Omron Sysmac Studio project delta_paper_0_2 (Sysmac Studio 1.54.0.64019, StandardProject)
(* parameteriaztion the n *)

# Controller new_Controller_0: NX1P2-1140DT version 1.18
Units and slaves: Node47 : MADLN05BE (E002); Node72 : MADLN05BE (E001); Node73 : MADLN05BE (E003)
Axis MC_Axis1, settings changed from default: AxisType=ServoType, UnitsConversion=EnumElement5, UnitsNumerator=8388608, UnitsDenominator=36, MaxVelocity=500, MaxJogVelocity=360, SoftwareLimitMode=ValidForSpecifiedValueImmediateStop, PositiveSoftwareLimit=75, NegativeSoftwareLimit=-29.2, OriginInputMode=EXT, StartDirection=NegativeDirection, OriginInputDetectionDirection=NegativeDirection, HomingVelocity=100, HomingApproachVelocity=10, HomingAcceleration=10, HomingDeceleration=20
Axis MC_Axis2, settings changed from default: AxisNumber=1, AxisType=ServoType, UnitsConversion=EnumElement5, UnitsNumerator=8388608, UnitsDenominator=36, MaxVelocity=500, MaxJogVelocity=360, SoftwareLimitMode=ValidForSpecifiedValueImmediateStop, PositiveSoftwareLimit=75, NegativeSoftwareLimit=-29.2
Axis MC_Axis3, settings changed from default: AxisNumber=2, AxisType=ServoType, UnitsConversion=EnumElement5, UnitsNumerator=8388608, UnitsDenominator=36, MaxVelocity=500, MaxJogVelocity=360, SoftwareLimitMode=ValidForSpecifiedValueDecreaseStop, PositiveSoftwareLimit=29.2, NegativeSoftwareLimit=-75
Task PrimaryTask (priority 4, period or condition 4000): Program0

TYPE InforRobot : STRUCT
    e : LREAL;
    rf : LREAL;
    re : LREAL;
    f : LREAL;
END_STRUCT END_TYPE
TYPE Input_Position : STRUCT
    X : LREAL;
    Y : LREAL;
    Z : LREAL;
END_STRUCT END_TYPE
TYPE Angle_Theta : STRUCT
    Theta1 : LREAL;
    Theta2 : LREAL;
    Theta3 : LREAL;
END_STRUCT END_TYPE
TYPE Bool_Theta : STRUCT
    Motor_Theta1 : REAL;
    Motor_Theta2 : REAL;
    Motor_Theta3 : REAL;
END_STRUCT END_TYPE
TYPE Speed_Theta : STRUCT
    Speed_Theta1 : REAL;
    Speed_Theta2 : REAL;
    Speed_Theta3 : REAL;
END_STRUCT END_TYPE
TYPE Workspace : STRUCT
    X_Min : REAL;
    X_Max : REAL;
    Y_Min : REAL;
    Y_Max : REAL;
    Z_Min : REAL;
    Z_Max : REAL;
END_STRUCT END_TYPE
TYPE From_pc : STRUCT
    n_points : INT;  (* new-> # of points *)
    commandID : INT;
    argument_number : INT;
    argument_x : ARRAY[0..31] OF real;
    argument_y : ARRAY[0..31] OF real;
    argument_z : ARRAY[0..31] OF real;
    argument_e : ARRAY[0..31] OF int;
    bit_doing : INT;
END_STRUCT END_TYPE
TYPE From_plc : STRUCT
    pos_angular : ARRAY[0..2] OF REAL;
    pos_EE : ARRAY[0..6] OF REAL;
    task_doing : INT;
    task_state : INT;
    Total_Time_Estimate : ARRAY[0..30] OF REAL;
    Total_Time_Sum : REAL;
    current_step : INT;
    n_points_ack : INT;
END_STRUCT END_TYPE

VAR_GLOBAL CONSTANT
    MC_Axis1 : _sAXIS_REF;  (* at MC://_MC_AX[0] *)
    MC_Axis2 : _sAXIS_REF;  (* at MC://_MC_AX[1] *)
    MC_Axis3 : _sAXIS_REF;  (* at MC://_MC_AX[2] *)
END_VAR
VAR_GLOBAL
    Out_Test0 : LREAL;
    Out_TestAngle1 : LREAL;
    Out_TestAngle2 : LREAL;
    Out_TestAngle3 : LREAL;
    MyHomingPara : _sHOMING_REF;
    Home_Axis1 : BOOL;  (* at BuiltInIO://cpu/#0/Input_Bit_00 *)
    Home_Axis2 : BOOL;  (* at BuiltInIO://cpu/#0/Input_Bit_01 *)
    Home_Axis3 : BOOL;  (* at BuiltInIO://cpu/#0/Input_Bit_02 *)
    Home_Lamp1 : BOOL;  (* at BuiltInIO://cpu/#0/Output_Bit_00 *)
    Home_Lamp2 : BOOL;  (* at BuiltInIO://cpu/#0/Output_Bit_01 *)
    Home_Lamp3 : BOOL;  (* at BuiltInIO://cpu/#0/Output_Bit_02 *)
    Out_Done_Inter : BOOL;
    pc_package : From_pc;  (* published *)
    plc_package : From_plc;  (* published *)
    Pump_Out : BOOL;  (* at BuiltInIO://cpu/#0/Output_Bit_03 *)
    Mc_On_Btn : BOOL;  (* at BuiltInIO://cpu/#0/Input_Bit_03 *)
    Res_Err_Btn : BOOL;  (* at BuiltInIO://cpu/#0/Input_Bit_04 *)
    Valve_Out : BOOL;  (* at BuiltInIO://cpu/#0/Output_Bit_04 *)
    Start_Home_Flag : BOOL;
    Home_Done_Flag1 : BOOL;
    Home_Done_Flag2 : BOOL;
    Home_Done_Flag3 : BOOL;
    button_teaching_ex : BOOL;  (* at BuiltInIO://cpu/#0/Input_Bit_06 *)
END_VAR
VAR_GLOBAL CONSTANT
    ICV_MAX_PT : UINT := 32;
END_VAR
VAR_GLOBAL
    ICV_n : INT := 4;
    ICV_Abort : BOOL;  (* Huy quy dao giua chung - noi tu Rung 1 E-Stop *)
    ICV_Err_Reset : BOOL;
    ICV_Pos_X : ARRAY[0..31] OF Lreal;
    ICV_Pos_Y : ARRAY[0..31] OF Lreal;
    ICV_Pos_Z : ARRAY[0..31] OF Lreal;
END_VAR

PROGRAM Program0
VAR
    Pw_servo_on : BOOL := False;
    MC_Move_Abs : BOOL;
    Pw_Power_0 : MC_Power;
    Pw_Power_1 : MC_Power;
    Pw_Power_2 : MC_Power;
    MC_Home_Ext : BOOL;  (* toggle 1 *)
    MC_Home_Delta_0 : MC_Home_Delta;
    Calib_Abs1 : MC_MoveAbsolute;
    Calib_Abs2 : MC_MoveAbsolute;
    Calib_Abs3 : MC_MoveAbsolute;
    Home_test_1 : MC_Home;
    Home_test_2 : MC_Home;
    Home_test_3 : MC_Home;
    X_cal : LREAL;
    Y_cal : LREAL;
    Z_cal : LREAL;
    pos_angular : LREAL;
    Goto_Abs : Goto_Absolute;
    when_it_turn2 : BOOL;
    Goto_abs_x : LREAL;
    Goto_abs_y : LREAL;
    Goto_abs_z : LREAL;
    another4 : BOOL;
    MC_Inter_Curve_Vel_0 : MC_Inter_Curve_Vel;
    MC_Inter_Curve_Vel_1 : MC_Inter_Curve_Vel;
    MC_Inter_Curve_Vel_2 : MC_Inter_Curve_Vel;
    MC_Inter_Curve_Vel_3 : MC_Inter_Curve_Vel;
    MC_Inter_Curve_Vel_4 : MC_Inter_Curve_Vel;
    MC_Inter_Curve_Vel_5 : MC_Inter_Curve_Vel;
    ICV_Start_NewTurn : BOOL;  (* Set 1 until ICV_Blend_done_2 *)
    ICV_Vmax : LREAL := 300;  (* 300 *)
    ICV_Amax : LREAL := 1000;  (* 1000 *)
    ICV_Dmax : LREAL := 1000;  (* 1000 *)
    Pump_Ext : BOOL;
    ICV_Pos_E : ARRAY[0..31] OF Int;
    ICV_t : ARRAY[0..30] OF Lreal;
    i1 : INT;
    MC_Goto_Abs : BOOL;  (* Set 1 until it done *)
    Fwk_Calc_OutX : REAL;
    Fwk_Calc_OutY : REAL;
    Fwk_Calc_OutZ : REAL;
    Moveto_Intermediary : MC_MoveAbsolute;
    Moveto_Midpoint : MC_MoveAbsolute;
    Moveto_Midpoint_1 : MC_MoveAbsolute;
    Moveto_Midpoint_2 : MC_MoveAbsolute;
    Moveto_Midpoint_3 : MC_MoveAbsolute;
    Home_Done : BOOL;
    Home_Error : BOOL;
    Goto_Abs_Error : BOOL;
    Pump_Res : BOOL;
    MC_ICV_Err : BOOL;
    MC_Stop1 : MC_Stop;
    MC_Stop2 : MC_Stop;
    MC_Stop3 : MC_Stop;
    MC_RES_DB1 : MC_Reset;
    MC_RES_DB2 : MC_Reset;
    MC_RES_DB3 : MC_Reset;
    Comment : BOOL;
    Mc_On_Btn_Flag : BOOL;
    Check_IK : BOOL;
    Goto_Abs2 : Goto_Absolute;
    Goto_Abs2_Exe : BOOL;
    Goto_Abs2_Done : BOOL;
    Out_TestAngle1_tmp : LREAL;
    Out_TestAngle2_tmp : LREAL;
    Out_TestAngle3_tmp : LREAL;
    Out_TestAngle10 : LREAL;
    Out_TestAngle20 : LREAL;
    Out_TestAngle30 : LREAL;
    Stop1 : MC_Power;
    MC_Stop4 : MC_Stop;
    MC_Stop5 : MC_Stop;
    MC_Stop6 : MC_Stop;
    Comment0 : BOOL;
    MC_Inter_Curve_Vel_6 : MC_Inter_Curve_Vel;
    ICV_Blend_Done_6 : BOOL;
    ICV_Vend_6 : LREAL;
    Current_Step : INT;
    fb_PumpTimer : TP;
    Var_Timer_IN : BOOL;
    Timing_for_EEF : TIME;
    i_t : INT;
    Mem_ICV_t5 : LREAL;
    k_t : LREAL;
    Teach_Index : INT := 0;  (* Chỉ số điểm học hiện tại (0..99) *)
    Teach_Max_Points : INT := 100;
    Teach_Array_X : ARRAY[0..99] OF LREAL := [100(0.0)];
    Teach_Array_Y : ARRAY[0..99] OF LREAL := [100(0.0)];
    Teach_Array_Z : ARRAY[0..99] OF LREAL := [100(0.0)];
    Teach_Array_Th1 : ARRAY[0..99] OF LREAL := [100(0.0)];
    Teach_Array_Th2 : ARRAY[0..99] OF LREAL := [100(0.0)];
    Teach_Array_Th3 : ARRAY[0..99] OF LREAL := [100(0.0)];
    Teach_Array_Full_E : BOOL;
    Teach_FB : FB_TeachingMode;
    button_teaching_active : BOOL;
    Traj : FB_ICV_Sequencer;
    ICV_Abort : BOOL := False;
    ICV_Err_Reset : BOOL := False;
    Mem_T_LastSeg : LREAL := 0.0;  (* Chot thoi gian doan cuoi cho bo dinh thoi bom *)
    Seq_LastSegReady : BOOL := False;  (* Doan cuoi VA da tinh xong thoi gian -> moi cho timer bom chay *)
END_VAR
VAR_EXTERNAL
    Out_Test0 : LREAL;
    Out_TestAngle1 : LREAL;
    Out_TestAngle2 : LREAL;
    Out_TestAngle3 : LREAL;
END_VAR
VAR_EXTERNAL CONSTANT
    MC_Axis1 : _sAXIS_REF;
    MC_Axis2 : _sAXIS_REF;
    MC_Axis3 : _sAXIS_REF;
END_VAR
VAR_EXTERNAL
    Home_Axis2 : BOOL;
    Home_Axis3 : BOOL;
    Out_Done_Inter : BOOL;
    plc_package : From_plc;
    pc_package : From_pc;
    Pump_Out : BOOL;
    Home_Axis1 : BOOL;
    Mc_On_Btn : BOOL;
    Res_Err_Btn : BOOL;
    Valve_Out : BOOL;
    Start_Home_Flag : BOOL;
    Home_Done_Flag1 : BOOL;
    Home_Done_Flag2 : BOOL;
    Home_Done_Flag3 : BOOL;
    button_teaching_ex : BOOL;
    ICV_Pos_X : ARRAY[0..31] OF Lreal;
    ICV_Pos_Y : ARRAY[0..31] OF Lreal;
    ICV_Pos_Z : ARRAY[0..31] OF Lreal;
    ICV_n : INT;
END_VAR
VAR
    _p1 : BOOL;
    _t2 : BOOL;
    _t3 : BOOL;
END_VAR

(* Section Section0: ladder, written here as Structured Text *)

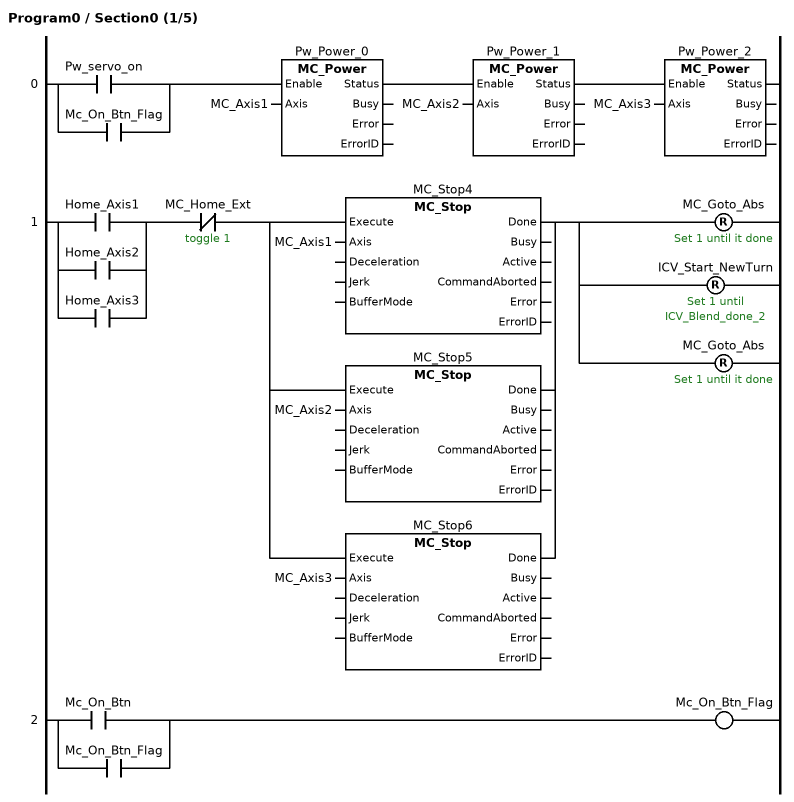
(* Rung 0 *)
Pw_Power_0(Enable := Pw_servo_on OR Mc_On_Btn_Flag, Axis := MC_Axis1);
Pw_Power_1(Enable := Pw_Power_0.Status, Axis := MC_Axis2);
Pw_Power_2(Enable := Pw_Power_1.Status, Axis := MC_Axis3);
(* Rung 1 *)
_p1 := (Home_Axis1 OR Home_Axis2 OR Home_Axis3) AND NOT MC_Home_Ext;
MC_Stop4(Execute := _p1, Axis := MC_Axis1);
MC_Stop5(Execute := _p1, Axis := MC_Axis2);
MC_Stop6(Execute := _p1, Axis := MC_Axis3);
IF MC_Stop4.Done OR MC_Stop5.Done OR MC_Stop6.Done THEN
    MC_Goto_Abs := FALSE;
    ICV_Start_NewTurn := FALSE;
    MC_Goto_Abs := FALSE;
END_IF;
(* Rung 2 *)
Mc_On_Btn_Flag := Mc_On_Btn OR Mc_On_Btn_Flag;

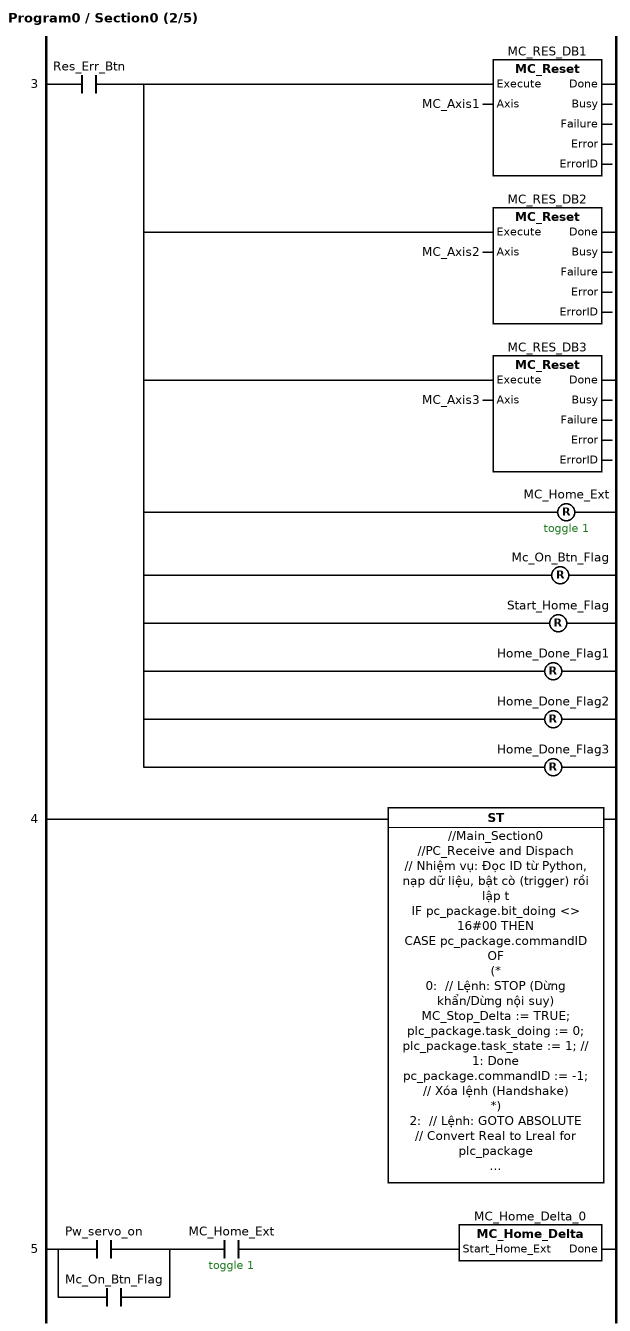
(* Rung 3 *)
MC_RES_DB1(Execute := Res_Err_Btn, Axis := MC_Axis1);
MC_RES_DB2(Execute := Res_Err_Btn, Axis := MC_Axis2);
MC_RES_DB3(Execute := Res_Err_Btn, Axis := MC_Axis3);
IF Res_Err_Btn THEN
    MC_Home_Ext := FALSE;
    Mc_On_Btn_Flag := FALSE;
    Start_Home_Flag := FALSE;
    Home_Done_Flag1 := FALSE;
    Home_Done_Flag2 := FALSE;
    Home_Done_Flag3 := FALSE;
END_IF;
(* Rung 4 *)
//Main_Section0 
//PC_Receive and Dispach
// Nhiệm vụ: Đọc ID từ Python, nạp dữ liệu, bật cò (trigger) rồi lập tức xóa ID

IF pc_package.bit_doing <> 16#00 THEN
CASE pc_package.commandID OF
  (*  
0:  // Lệnh: STOP (Dừng khẩn/Dừng nội suy)
	        MC_Stop_Delta := TRUE;
	        
	        plc_package.task_doing := 0;
	        plc_package.task_state := 1; // 1: Done
	        pc_package.commandID := -1;  // Xóa lệnh (Handshake)
			*)
    2:  // Lệnh: GOTO ABSOLUTE
		// Convert Real to Lreal for plc_package
		Goto_abs_x:= REAL_TO_LREAL(pc_package.argument_x[0]);
		Goto_abs_y := REAL_TO_LREAL(pc_package.argument_y[0]);
		Goto_abs_z:= REAL_TO_LREAL(pc_package.argument_z[0]);
        
        MC_Goto_Abs := TRUE;         // Bật cò chạy
        plc_package.task_doing := 2;
        plc_package.task_state := 2; // 2: Busy
        pc_package.commandID := -1;

    3:  // Lệnh: GO TRAJECTORY (Chạy quỹ đạo theo mảng tọa độ)
        ICV_Start_NewTurn := TRUE; //auto turn off
        FOR i1 := 0 TO 6 DO
			ICV_Pos_X[i1] := REAL_TO_LREAL(pc_package.argument_x[i1]);
			ICV_Pos_Y[i1] := REAL_TO_LREAL(pc_package.argument_y[i1]);
			ICV_Pos_Z[i1] := REAL_TO_LREAL(pc_package.argument_z[i1]);
			ICV_Pos_E[i1] := pc_package.argument_e[i1];
		END_FOR;
        plc_package.task_doing := 3;
        plc_package.task_state := 2; // Busy
        pc_package.commandID := -1;

    4:  // Lệnh: HOME CALIBRATION (Tìm gốc)
        MC_Home_Ext := TRUE;
        
        plc_package.task_doing := 4;
        plc_package.task_state := 2; // Busy
        pc_package.commandID := -1;

    5:  // Lệnh: PICK (Hút vật)
        Pump_Ext := TRUE;
        
        plc_package.task_doing := 5;
        plc_package.task_state := 1; // 1: Done (Do bật bơm là xong ngay)
        pc_package.commandID := -1;

    6:  // Lệnh: RELEASE (Nhả vật)
        Pump_Ext := FALSE;
        
        plc_package.task_doing := 6;
        plc_package.task_state := 1; // Done
        pc_package.commandID := -1;
		END_CASE;
pc_package.bit_doing :=16#00;
END_IF;
(* Rung 5 *)
MC_Home_Delta_0(Start_Home_Ext := (Pw_servo_on OR Mc_On_Btn_Flag) AND MC_Home_Ext);

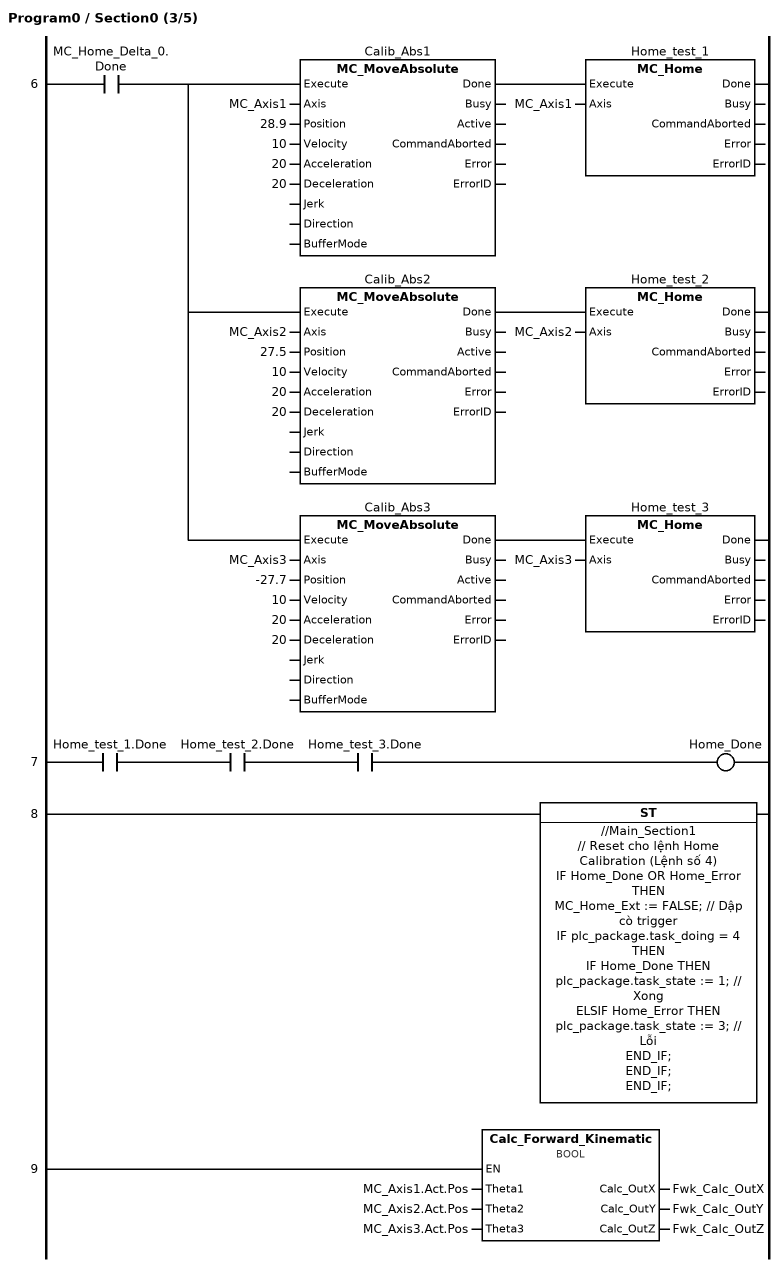
(* Rung 6 *)
Calib_Abs1(Execute := MC_Home_Delta_0.Done, Axis := MC_Axis1, Position := 28.9, Velocity := 10, Acceleration := 20, Deceleration := 20);
Home_test_1(Execute := Calib_Abs1.Done, Axis := MC_Axis1);
Calib_Abs2(Execute := MC_Home_Delta_0.Done, Axis := MC_Axis2, Position := 27.5, Velocity := 10, Acceleration := 20, Deceleration := 20);
Home_test_2(Execute := Calib_Abs2.Done, Axis := MC_Axis2);
Calib_Abs3(Execute := MC_Home_Delta_0.Done, Axis := MC_Axis3, Position := -27.7, Velocity := 10, Acceleration := 20, Deceleration := 20);
Home_test_3(Execute := Calib_Abs3.Done, Axis := MC_Axis3);
(* Rung 7 *)
Home_Done := Home_test_1.Done AND Home_test_2.Done AND Home_test_3.Done;
(* Rung 8 *)
//Main_Section1 
// Reset cho lệnh Home Calibration (Lệnh số 4)
IF Home_Done OR Home_Error THEN
 
    MC_Home_Ext := FALSE; // Dập cò trigger
	
    IF plc_package.task_doing = 4 THEN
        IF Home_Done THEN
            plc_package.task_state := 1; // Xong
        ELSIF Home_Error THEN
            plc_package.task_state := 3; // Lỗi
        END_IF;
    END_IF;
    
END_IF;
(* Rung 9 *)
_t2 := Calc_Forward_Kinematic(Theta1 := MC_Axis1.Act.Pos, Theta2 := MC_Axis2.Act.Pos, Theta3 := MC_Axis3.Act.Pos, Calc_OutX => Fwk_Calc_OutX, Calc_OutY => Fwk_Calc_OutY, Calc_OutZ => Fwk_Calc_OutZ);

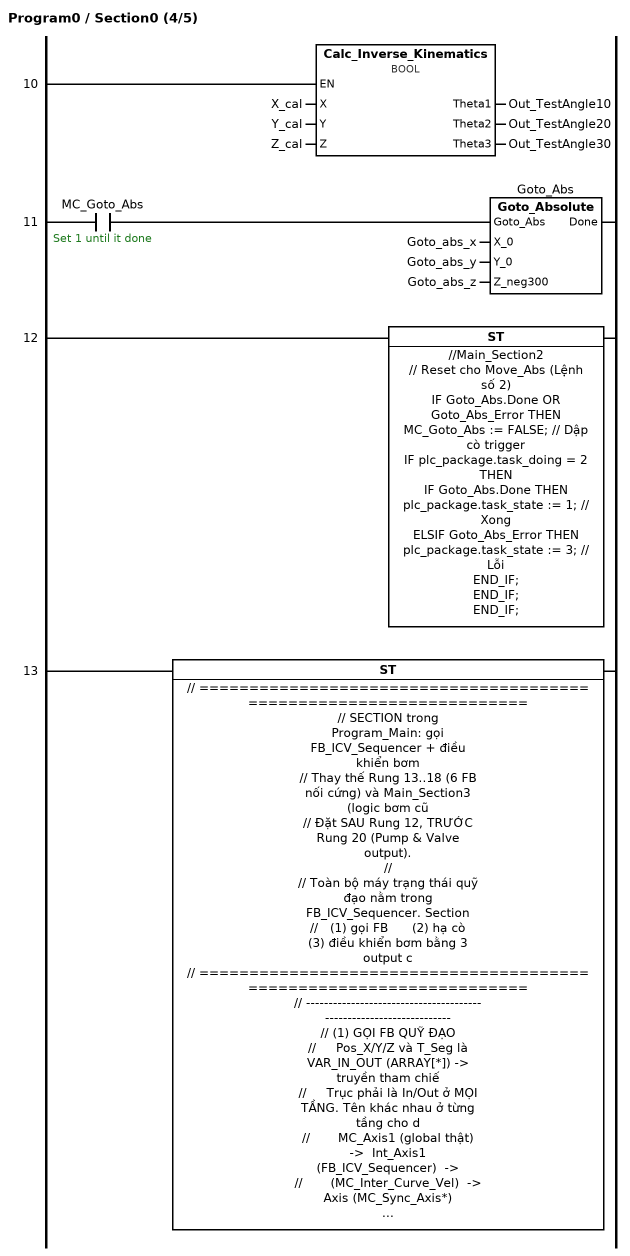
(* Rung 10 *)
_t3 := Calc_Inverse_Kinematics(X := X_cal, Y := Y_cal, Z := Z_cal, Theta1 => Out_TestAngle10, Theta2 => Out_TestAngle20, Theta3 => Out_TestAngle30);
(* Rung 11 *)
Goto_Abs(Goto_Abs := MC_Goto_Abs, X_0 := Goto_abs_x, Y_0 := Goto_abs_y, Z_neg300 := Goto_abs_z);
(* Rung 12 *)
//Main_Section2
// Reset cho Move_Abs (Lệnh số 2)
IF Goto_Abs.Done OR Goto_Abs_Error THEN
 
    MC_Goto_Abs := FALSE; // Dập cò trigger
	
    IF plc_package.task_doing = 2 THEN
        IF Goto_Abs.Done THEN
            plc_package.task_state := 1; // Xong
        ELSIF Goto_Abs_Error THEN
            plc_package.task_state := 3; // Lỗi
        END_IF;
    END_IF;
    
END_IF;
(* Rung 13 *)
// =====================================================================================
// SECTION trong Program_Main: gọi FB_ICV_Sequencer + điều khiển bơm
// Thay thế Rung 13..18 (6 FB nối cứng) và Main_Section3 (logic bơm cũ).
// Đặt SAU Rung 12, TRƯỚC Rung 20 (Pump & Valve output).
//
// Toàn bộ máy trạng thái quỹ đạo nằm trong FB_ICV_Sequencer. Section này chỉ:
//   (1) gọi FB      (2) hạ cò      (3) điều khiển bơm bằng 3 output của FB
// =====================================================================================


// -------------------------------------------------------------------------------------
// (1) GỌI FB QUỸ ĐẠO
//     Pos_X/Y/Z và T_Seg là VAR_IN_OUT (ARRAY[*]) -> truyền tham chiếu, KHÔNG copy mảng.
//     Trục phải là In/Out ở MỌI TẦNG. Tên khác nhau ở từng tầng cho dễ phân biệt:
//       MC_Axis1 (global thật)  ->  Int_Axis1 (FB_ICV_Sequencer)  ->  MC_Axis1
//       (MC_Inter_Curve_Vel)  ->  Axis (MC_Sync_Axis*)
// -------------------------------------------------------------------------------------
Traj(
    Execute  := ICV_Start_NewTurn,
    Abort    := ICV_Abort,
    ErrReset := ICV_Err_Reset,
    N_Points := ICV_n,
    Max_Index:= 31,                 // chỉ số lớn nhất của ICV_Pos_X (ARRAY[0..31])
    V_max    := ICV_Vmax,
    A_max    := ICV_Amax,
    D_max    := ICV_Dmax,
    Pos_X    := ICV_Pos_X,
    Pos_Y    := ICV_Pos_Y,
    Pos_Z    := ICV_Pos_Z,
    T_Seg    := ICV_t,
    // TRÁI = tên tham số của FB_ICV_Sequencer ; PHẢI = biến global của trục thật
    Int_Axis1:= MC_Axis1,
    Int_Axis2:= MC_Axis2,
    Int_Axis3:= MC_Axis3
);


// -------------------------------------------------------------------------------------
// (2) HẠ CÒ NGAY SAU LỜI GỌI
//     FB đã bắt SƯỜN LÊN của Execute ở khối (1) rồi, nên hạ ngay là an toàn.
//
//     KHÔNG dùng "IF Traj.Busy THEN": khi FB TỪ CHỐI lệnh (N_Points sai -> ErrorID = 1)
//     thì Busy KHÔNG BAO GIỜ lên TRUE -> cò kẹt TRUE vĩnh viễn -> mọi lệnh sau đó không
//     tạo được sườn lên nữa -> quỹ đạo chết hẳn, phải khởi động lại PLC.
// -------------------------------------------------------------------------------------
IF ICV_Start_NewTurn THEN
    ICV_Start_NewTurn := FALSE;
END_IF;

// Xoá cờ ErrReset sau 1 chu kỳ (nút Res_Err_Btn có thể bị giữ lâu)
IF ICV_Err_Reset AND NOT Traj.Error THEN
    ICV_Err_Reset := FALSE;
END_IF;


// -------------------------------------------------------------------------------------
// (3) ĐIỀU KHIỂN BƠM / END-EFFECTOR
//     Đoạn 0 .. n-3 : bơm bám theo ICV_Pos_E[SegIdx]
//     Đoạn cuối     : bơm nhả sớm ở 50% thời gian đoạn, cho vật kịp rơi trước khi tay đi
// -------------------------------------------------------------------------------------

// "Đoạn cuối SẴN SÀNG" = đang ở đoạn cuối VÀ FB đã tính xong thời gian của đoạn đó.
//
// PHẢI chờ T_SegNow > 0. Ngay chu kỳ vừa chuyển sang đoạn cuối, Out_T_Segment của
// MC_Inter_Curve_Vel VẪN ĐANG GIỮ thời gian của đoạn TRƯỚC (nó chỉ bị xoá ở State 0
// của đoạn mới, tức chu kỳ sau). Chốt vội sẽ lấy nhầm số của đoạn trước.
Seq_LastSegReady := Traj.IsLastSeg AND (Traj.T_SegNow > 0.0);

IF Seq_LastSegReady THEN
    Mem_T_LastSeg := Traj.T_SegNow;
END_IF;

Timing_for_EEF := NanoSecToTime(LREAL_TO_LINT(0.5 * Mem_T_LastSeg * 1000000000.0));

// IN dùng Seq_LastSegReady, KHÔNG dùng Traj.IsLastSeg.
// TP chốt PT tại SƯỜN LÊN của IN -> phải đợi PT đúng rồi mới cho timer chạy.
// Trễ 2 chu kỳ (8 ms) so với đầu đoạn cuối, không đáng kể.
fb_PumpTimer(IN := Seq_LastSegReady, PT := Timing_for_EEF);

IF NOT Traj.Busy THEN
    Pump_Ext := FALSE;

ELSIF Traj.IsLastSeg THEN
    // GIỮ NGUYÊN biểu thức của code cũ: đúng khi fb_PumpTimer khai báo là TP (Pulse).
    //   TP  -> .Q = TRUE trong 50% đầu, tự hạ sau đó -> bơm nhả ở giữa đoạn.  ĐÚNG
    //   TON -> .Q = FALSE trong 50% đầu -> bơm chỉ bật ở nửa SAU. NGƯỢC Ý ĐỒ.
    // Nếu instance đang là TON, đổi thành:  AND NOT fb_PumpTimer.Q
    //
    // "OR NOT Seq_LastSegReady" giữ bơm ON trong 2 chu kỳ chờ timer khởi động,
    // tránh hụt chân không 8 ms ngay đầu đoạn cuối.
    Pump_Ext := (ICV_Pos_E[Traj.SegIdx] = 1)
                AND (fb_PumpTimer.Q OR NOT Seq_LastSegReady);

ELSE
    Pump_Ext := (ICV_Pos_E[Traj.SegIdx] = 1);
END_IF;

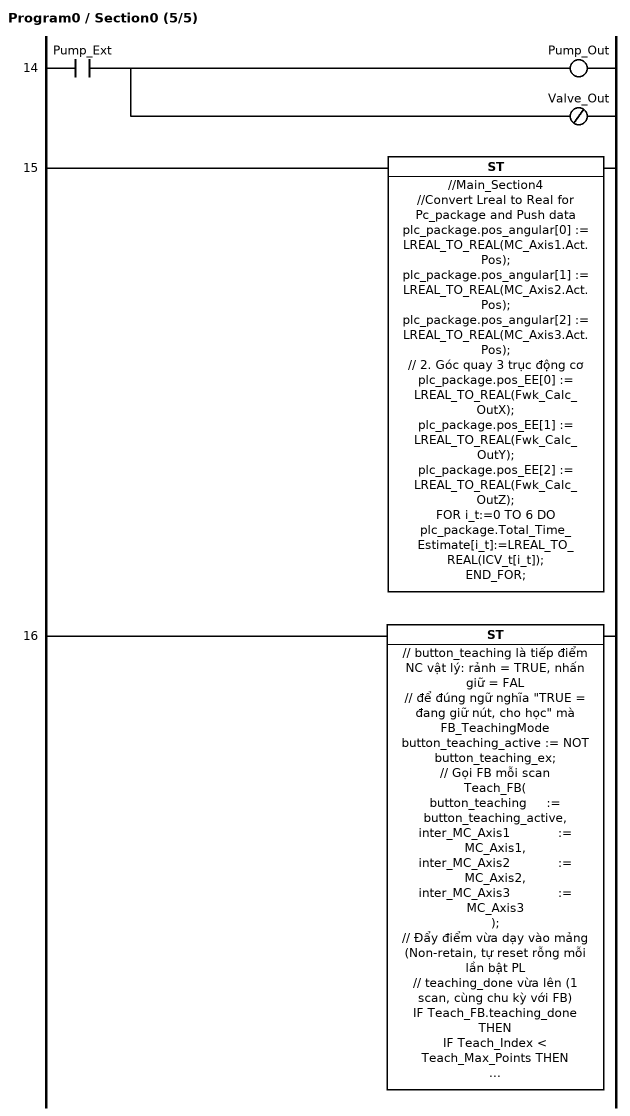
(* Rung 14 *)
Pump_Out := Pump_Ext;
Valve_Out := NOT Pump_Ext;
(* Rung 15 *)
//Main_Section4
//Convert Lreal to Real for Pc_package and Push data
plc_package.pos_angular[0] := LREAL_TO_REAL(MC_Axis1.Act.Pos);
plc_package.pos_angular[1] := LREAL_TO_REAL(MC_Axis2.Act.Pos);
plc_package.pos_angular[2] := LREAL_TO_REAL(MC_Axis3.Act.Pos);

// 2. Góc quay 3 trục động cơ
plc_package.pos_EE[0] := LREAL_TO_REAL(Fwk_Calc_OutX); 
plc_package.pos_EE[1] := LREAL_TO_REAL(Fwk_Calc_OutY); 
plc_package.pos_EE[2] := LREAL_TO_REAL(Fwk_Calc_OutZ);

FOR i_t:=0 TO 6 DO
	plc_package.Total_Time_Estimate[i_t]:=LREAL_TO_REAL(ICV_t[i_t]);
END_FOR;
(* Rung 16 *)
// button_teaching là tiếp điểm NC vật lý: rảnh = TRUE, nhấn giữ = FALSE -> đảo lại
// để đúng ngữ nghĩa "TRUE = đang giữ nút, cho học" mà FB_TeachingMode yêu cầu.
button_teaching_active := NOT button_teaching_ex;

// Gọi FB mỗi scan
Teach_FB(
    button_teaching     := button_teaching_active,
    inter_MC_Axis1            := MC_Axis1,
    inter_MC_Axis2            := MC_Axis2,
    inter_MC_Axis3            := MC_Axis3	
);

// Đẩy điểm vừa dạy vào mảng (Non-retain, tự reset rỗng mỗi lần bật PLC) — chỉ khi
// teaching_done vừa lên (1 scan, cùng chu kỳ với FB)
IF Teach_FB.teaching_done THEN
    IF Teach_Index < Teach_Max_Points THEN
        Teach_Array_X[Teach_Index]   := Teach_FB.pos_teaching1;
        Teach_Array_Y[Teach_Index]   := Teach_FB.pos_teaching2;
        Teach_Array_Z[Teach_Index]   := Teach_FB.pos_teaching3;
        Teach_Array_Th1[Teach_Index] := LREAL_TO_REAL(Teach_FB.theta_teaching1);
        Teach_Array_Th2[Teach_Index] := LREAL_TO_REAL(Teach_FB.theta_teaching2);
        Teach_Array_Th3[Teach_Index] := LREAL_TO_REAL(Teach_FB.theta_teaching3);
        Teach_Index := Teach_Index + 1;
        Teach_Array_Full_E := FALSE;
    ELSE
        // Mảng đã đầy: không có chỗ lưu, báo lỗi rõ ràng thay vì âm thầm bỏ qua
        Teach_Array_Full_E := TRUE;
    END_IF;
END_IF;

// HMI / Python PC (poll chậm qua TCP/IP) nên theo dõi Teach_Index tăng dần
// thay vì bắt xung teaching_done — tránh miss tín hiệu do chu kỳ poll không đồng bộ scan PLC.
END_PROGRAM

FUNCTION Calc_Inverse_Kinematics : BOOL
VAR CONSTANT
    Cos120 : LREAL := -0.5;
    Sin120 : LREAL := 0.8660254037844386;
END_VAR
VAR
    tmp_Theta1 : LREAL;
    tmp_Theta2 : LREAL;
    tmp_Theta3 : LREAL;
    rotate_X2 : LREAL;
    rotate_Y2 : LREAL;
    rotate_X3 : LREAL;
    rotate_Y3 : LREAL;
END_VAR
VAR CONSTANT
    rf : LREAL := 346.4;
    re : LREAL := 86.6;
    f : LREAL := 140;
    e : LREAL := 315;
END_VAR
VAR
    Out_Error_IK : BOOL;
END_VAR
VAR_INPUT
    X : LREAL;
    Y : LREAL;
    Z : LREAL;
END_VAR
VAR_OUTPUT
    Theta1 : LREAL;
    Theta2 : LREAL;
    Theta3 : LREAL;
END_VAR
// Khởi tạo lại cờ báo lỗi ở mỗi đầu chu kỳ quét (Primary Task)
Out_Error_IK := FALSE;

// -----------------------------------------------------------------------
// TÍNH TOÁN THETA 1 (Cánh tay 1 - Không xoay trục)
// -----------------------------------------------------------------------
Calc_Inverse_Kinematics := Calc_Angles_YZ(
    X0 := X, 
    Y0 := Y, 
    Z0 := Z,
    OutTheta => tmp_Theta1
);

	
// [TỐI ƯU B] Xử lý lỗi an toàn: Nếu tính toán IK thất bại (Tọa độ ngoài tầm với)
IF Calc_Inverse_Kinematics = TRUE  OR tmp_Theta1 <-20 THEN
    Out_Error_IK := TRUE; // Bật cờ báo lỗi ra hệ thống
    RETURN;               // Ngắt tính toán ngay lập tức
END_IF;

// [TỐI ƯU A] Truyền thẳng giá trị LREAL nguyên bản xuống Servo, BỎ HÀM ROUND
Theta1 := tmp_Theta1;


// -----------------------------------------------------------------------
// TÍNH TOÁN THETA 2 (Cánh tay 2 - Xoay hệ tọa độ đi -120 độ)
// -----------------------------------------------------------------------
rotate_X2 := X * Cos120 + Y * Sin120;
rotate_Y2 := Y * Cos120 - X * Sin120;

Calc_Inverse_Kinematics := Calc_Angles_YZ(
    X0 := rotate_X2, 
    Y0 := rotate_Y2, 
    Z0 := Z,
    OutTheta => tmp_Theta2
);

IF Calc_Inverse_Kinematics = TRUE OR tmp_Theta2 <-20 THEN
    Out_Error_IK := TRUE;
    RETURN;
END_IF;

Theta2 := tmp_Theta2;


// -----------------------------------------------------------------------
// TÍNH TOÁN THETA 3 (Cánh tay 3 - Xoay hệ tọa độ đi +120 độ)
// -----------------------------------------------------------------------
rotate_X3 := X * Cos120 - Y * Sin120;
rotate_Y3 := Y * Cos120 + X * Sin120;

Calc_Inverse_Kinematics := Calc_Angles_YZ(
    X0 := rotate_X3, 
    Y0 := rotate_Y3, 
    Z0 := Z,
    OutTheta => tmp_Theta3
);

IF Calc_Inverse_Kinematics = TRUE OR tmp_Theta3*-1 >20 THEN
    Out_Error_IK := TRUE;
    RETURN;
END_IF;

Theta3 := tmp_Theta3*-1;
END_FUNCTION

FUNCTION Calc_Angles_YZ : BOOL  (* return true -> False in inverse calc *)
VAR
    tmp_y0 : LREAL;
    a : LREAL;
    b : LREAL;
    d : LREAL;
    yj : LREAL;
    zj : LREAL;
    y1 : LREAL;
    tmp_AnglePi : LREAL;
END_VAR
VAR CONSTANT
    Pi : LREAL := 3.141592653589793;
    Tan30 : LREAL := 0.5773502691896257;
    Base : LREAL := 346.4;
    EndEffector : LREAL := 86.6;
    Bicep : LREAL := 140;
    Forearm : LREAL := 315;
END_VAR
VAR_INPUT
    X0 : LREAL;
    Y0 : LREAL;
    Z0 : LREAL;
END_VAR
VAR_OUTPUT
    OutTheta : LREAL;
END_VAR
(*
// FUNCTION: Calc_Angles_YZ (Cal the inverse in 2D-space)
//All variants use Lreal to uttilize the precision of servo and syns all data

// [] Bẫy lỗi chia cho 0: Nếu tọa độ Z0 = 0 (End-effector nằm ngang với Base)
// Phép tính 'a' và 'b' bên dưới sẽ bị lỗi chia cho 0 làm CPU PLC báo lỗi (Major Fault)
*)
IF Z0 = 0.0 THEN
    Calc_Angles_YZ := TRUE; // turn Error true
    RETURN;
END_IF;

// Calc the Y1 and have temp_y0 (the prosition of the Y0 with Y1)
y1 := -0.5 * Tan30* Base;   // the point of edge of fix-triangle
tmp_y0 := Y0 - (0.5 *Tan30* EndEffector);  // the point of the edge of active-triagle

// we have ellbow (0,yj,zj) is contraint with:
//1. on a circle (0,y1,0) with R = bicep so (yj-y1)^2 + z_j^2 = bicep^2
//2. distance from End-effector (X0, tmp_y0,z0) equal the Forearm so
// X0^2 + (tmp_y0 - yj)^2 + (z-zj)^2 = forearm^2
// mathemitical tranformation we have linear function z with a and b bellow
// zj = a + b*yj => we have zj and we tranfer it to equation 1 and solve the two level function with yj
a := (X0*X0 + tmp_y0 * tmp_y0 + Z0 * Z0 + Bicep * Bicep - Forearm * Forearm - y1 * y1) / (2.0 * Z0);
b := (y1 - tmp_y0) / Z0;

// the delta of two level function with yj
d := - (a + b * y1) * (a + b * y1) + Bicep * (b * b * Bicep + Bicep);

// Kiểm tra xem điểm có tồn tại trong vùng không gian (Workspace) không
IF d < 0.0 THEN
    Calc_Angles_YZ := TRUE; // Trả về lỗi (Điểm không với tới được)
    RETURN;
END_IF;

yj := (y1 - a * b - SQRT(d)) / (b * b + 1.0);
zj := a + b * yj;

tmp_AnglePi := 0.0;
IF yj > y1 THEN
    tmp_AnglePi := 180.0;
END_IF;

// [TỐI ƯU 3] Bẫy lỗi chia cho 0 trong hàm tính góc ATAN
// Khi y1 = yj, phép chia (-zj / (y1 - yj)) sẽ gây lỗi PLC
IF (y1 - yj) = 0.0 THEN
    IF -zj >= 0.0 THEN
        OutTheta := 90.0 + tmp_AnglePi;
    ELSE
        OutTheta := -90.0 + tmp_AnglePi;
    END_IF;
ELSE
    // Tính góc Theta. Sử dụng hằng số '_pi' có sẵn của Sysmac Studio
    OutTheta := 180.0 * ATAN(-zj / (y1 - yj)) / Pi + tmp_AnglePi;
END_IF;

// Trả về FALSE khi tính toán thành công
Calc_Angles_YZ := FALSE;
RETURN;
END_FUNCTION

FUNCTION Calc_Forward_Kinematic : BOOL
VAR
    w : LREAL;
    Cos30 : LREAL := 0.8660254037844386;
    Pi : LREAL := 3.141592653589793;
    Tan30 : LREAL := 0.5773502691896257;
    Sin30 : LREAL := 0.5;
END_VAR
VAR CONSTANT
    Base : LREAL := 346.4;
    EndEffector : LREAL := 86.6;
    Bicep : LREAL := 140;
    Forearm : LREAL := 315;
END_VAR
VAR
    x_j1 : LREAL;
    y_j1 : LREAL;
    z_j1 : LREAL;
    x_j2 : LREAL;
    y_j2 : LREAL;
    z_j2 : LREAL;
    x_j3 : LREAL;
    y_j3 : LREAL;
    z_j3 : LREAL;
    r1 : LREAL;
    r2 : LREAL;
    r3 : LREAL;
    a1 : LREAL;
    a2 : LREAL;
    b1 : LREAL;
    b2 : LREAL;
    demon : LREAL;
    A_quad : LREAL;
    B_quad : LREAL;
    C_quad : LREAL;
    d : LREAL;
    t3 : LREAL;
    t2 : LREAL;
    t1 : LREAL;
    Calc_Forward_Kinematics : BOOL;
    OutX : LREAL;
    OutZ : LREAL;
    OutY : LREAL;
    D1_coeff : LREAL;
    A1_coeff : LREAL;
    B1_coeff : LREAL;
    C1_coeff : LREAL;
    A2_coeff : LREAL;
    B2_coeff : LREAL;
    C2_coeff : LREAL;
    D2_coeff : LREAL;
    det : LREAL;
END_VAR
VAR_INPUT
    Theta1 : LREAL;
    Theta2 : LREAL;
    Theta3 : LREAL;
END_VAR
VAR_OUTPUT
    Calc_OutX : REAL;
    Calc_OutY : REAL;
    Calc_OutZ : REAL;
END_VAR
VAR_EXTERNAL CONSTANT
    MC_Axis1 : _sAXIS_REF;
    MC_Axis2 : _sAXIS_REF;
    MC_Axis3 : _sAXIS_REF;
END_VAR
// =======================================================================
// FUNCTION: Calc_Forward_Kinematics (Tính toán động học thuận Robot Delta 3D)
// Trả về FALSE nếu tính toán thành công, TRUE nếu điểm nằm ngoài vùng làm việc
// =======================================================================
// LẤY GIÁ TRỊ GÓC THỰC TẾ (ACTUAL POSITION) TỪ ENCODER CỦA TRỤC
// =======================================================================
// Chuyển đổi các góc hiện tại từ Độ sang Radian
t1 := Theta1 * Pi / 180.0;
t2 := Theta2 * Pi / 180.0;
t3 := Theta3 * Pi / -180.0;

// Tính toán độ lệch tâm tương đối giữa Base và EndEffector
// (w chính là dịch tâm ngang từ gốc tọa độ đến khớp khuỷu tay nếu chiếu lên mặt phẳng XY)
w := 0.5 * Tan30 * (Base - EndEffector);

// =======================================================================
// BƯỚC 1: Tìm tọa độ không gian (x, y, z) của 3 khớp khuỷu tay (Elbow Joints)
// Hệ tọa độ tiêu chuẩn: Trục 1 nằm dọc theo phần âm của trục Y
// =======================================================================

// Trục 1 (Góc lệch 0 độ so với trục tính toán, xoay về -Y)
x_j1 := 0.0;
y_j1 := -(w + Bicep * COS(t1));
z_j1 := -Bicep * SIN(t1);

// Trục 2 (Xoay +120 độ)
x_j2 := (w + Bicep * COS(t2)) * Cos30;
y_j2 := (w + Bicep * COS(t2)) * Sin30;
z_j2 := -Bicep * SIN(t2);

// Trục 3 (Xoay -120 độ hoặc 240 độ)
x_j3 := -(w + Bicep * COS(t3)) * Cos30;
y_j3 := (w + Bicep * COS(t3)) * Sin30;
z_j3 := -Bicep * SIN(t3);

// =======================================================================
// BƯỚC 2: Giải hệ 3 phương trình mặt cầu có tâm tại các Elbow, bán kính Forearm
// =======================================================================

// =======================================================================
// BƯỚC 2: Giải hệ 3 phương trình mặt cầu (Dạng tổng quát, KHÔNG RÚT GỌN SAI)
// =======================================================================
// BƯỚC 2: Giải hệ 3 phương trình mặt cầu có tâm tại các Elbow (Phiên bản Tổng quát)
// =======================================================================

// Tính tổng bình phương tọa độ của các Elbow
r1 := y_j1 * y_j1 + z_j1 * z_j1;  // x_j1 = 0
r2 := x_j2 * x_j2 + y_j2 * y_j2 + z_j2 * z_j2;
r3 := x_j3 * x_j3 + y_j3 * y_j3 + z_j3 * z_j3;

// Thiết lập các hệ số cho hệ phương trình tuyến tính 2 ẩn (X, Y) theo tham số Z
// Dạng: 
// A1*X + B1*Y = D1 - C1*Z
// A2*X + B2*Y = D2 - C2*Z

A1_coeff := x_j2;                   // Thực chất là (x_j2 - x_j1) nhưng x_j1 = 0
B1_coeff := y_j2 - y_j1;
C1_coeff := z_j2 - z_j1;
D1_coeff := 0.5 * (r2 - r1);

A2_coeff := x_j3;                   // Thực chất là (x_j3 - x_j1) nhưng x_j1 = 0
B2_coeff := y_j3 - y_j1;
C2_coeff := z_j3 - z_j1;
D2_coeff := 0.5 * (r3 - r1);

// Tính định thức (Determinant) của hệ phương trình
det := (A1_coeff * B2_coeff) - (A2_coeff * B1_coeff);

// Bẫy lỗi: Hệ vô nghiệm (Chỉ xảy ra khi 3 khuỷu tay cùng nằm trên 1 đường thẳng)
IF det = 0.0 THEN
    Calc_Forward_Kinematics := TRUE; 
    RETURN;
END_IF;

// Sử dụng quy tắc Cramer để tìm a1, b1 (Cho X) và a2, b2 (Cho Y)
// Để biểu diễn: X0 = a1 + b1*Z0
a1 := (D1_coeff * B2_coeff - D2_coeff * B1_coeff) / det;
b1 := -(C1_coeff * B2_coeff - C2_coeff * B1_coeff) / det;

// Để biểu diễn: Y0 = a2 + b2*Z0
a2 := (A1_coeff * D2_coeff - A2_coeff * D1_coeff) / det;
b2 := -(A1_coeff * C2_coeff - A2_coeff * C1_coeff) / det;

// =======================================================================
// BƯỚC 3: Thay X0, Y0 vào phương trình mặt cầu 1 để tìm Z0
// Tạo thành phương trình bậc 2: A_quad * Z0^2 + B_quad * Z0 + C_quad = 0
// =======================================================================

A_quad := b1 * b1 + b2 * b2 + 1.0;
B_quad := 2.0 * (a1 * b1 + a2 * b2 - b2 * y_j1 - z_j1);
C_quad := a1 * a1 + a2 * a2 - 2.0 * a2 * y_j1 + r1 - (Forearm * Forearm);

// Tính Delta (Discriminant)
d := (B_quad * B_quad) - (4.0 * A_quad * C_quad);

// Kiểm tra xem vị trí các góc hiện tại có tạo ra tọa độ hợp lệ không
IF d < 0.0 THEN
    Calc_Forward_Kinematics := TRUE; // Trả về lỗi: Các khớp không thể kết nối
    RETURN;
END_IF;

// Tính tọa độ trung tâm End-Effector (Z lấy nghiệm có dấu trừ phía trước SQRT 
// vì đặc thù cơ cấu Delta robot làm việc ở nửa dưới trục Z)
OutZ := (-B_quad - SQRT(d)) / (2.0 * A_quad);

// Đẩy ngược Z0 vào hệ số tuyến tính để tìm X0 và Y0
OutX := a1 + b1 * OutZ;
OutY := a2 + b2 * OutZ;

Calc_OutZ := LREAL_TO_REAL(OutZ);
Calc_OutX := LREAL_TO_REAL(a1 + b1 * OutZ);
Calc_OutY := LREAL_TO_REAL(a2 + b2 * OutZ);

// Tính toán thành công
Calc_Forward_Kinematics := FALSE;
RETURN;
END_FUNCTION

FUNCTION_BLOCK MC_Home_Delta
VAR
    Move_Vel_Axis1 : MC_MoveVelocity;
    Start_Home : BOOL;
    MC_Stop_Axis1 : MC_Stop;
    Move_Vel_Axis2 : MC_MoveVelocity;
    Move_Vel_Axis3 : MC_MoveVelocity;
    MC_Stop_Axis2 : MC_Stop;
    MC_Stop_Axis3 : MC_Stop;
    MC_Home_Axis1 : MC_Home;
    MC_Home_Axis2 : MC_Home;
    MC_Home_Axis3 : MC_Home;
    t_home : TON;
    t2 : TON;
    t1 : TON;
    t3 : TON;
    TP1 : TP;
    TP2 : TP;
    TP4 : TP;
END_VAR
VAR_INPUT
    Start_Home_Ext : BOOL;
END_VAR
VAR_OUTPUT
    Done : BOOL;
END_VAR
VAR_EXTERNAL
    Home_Axis1 : BOOL;
    Home_Axis2 : BOOL;
    Home_Axis3 : BOOL;
END_VAR
VAR_EXTERNAL CONSTANT
    MC_Axis3 : _sAXIS_REF;
    MC_Axis2 : _sAXIS_REF;
    MC_Axis1 : _sAXIS_REF;
END_VAR
VAR_EXTERNAL
    Home_Lamp3 : BOOL;
    Home_Lamp1 : BOOL;
    Home_Lamp2 : BOOL;
    Start_Home_Flag : BOOL;
    Home_Done_Flag1 : BOOL;
    Home_Done_Flag2 : BOOL;
    Home_Done_Flag3 : BOOL;
END_VAR
VAR
    _e1 : R_TRIG;
    _e2 : R_TRIG;
    _e3 : R_TRIG;
    _e4 : R_TRIG;
END_VAR
(* ladder, written here as Structured Text *)

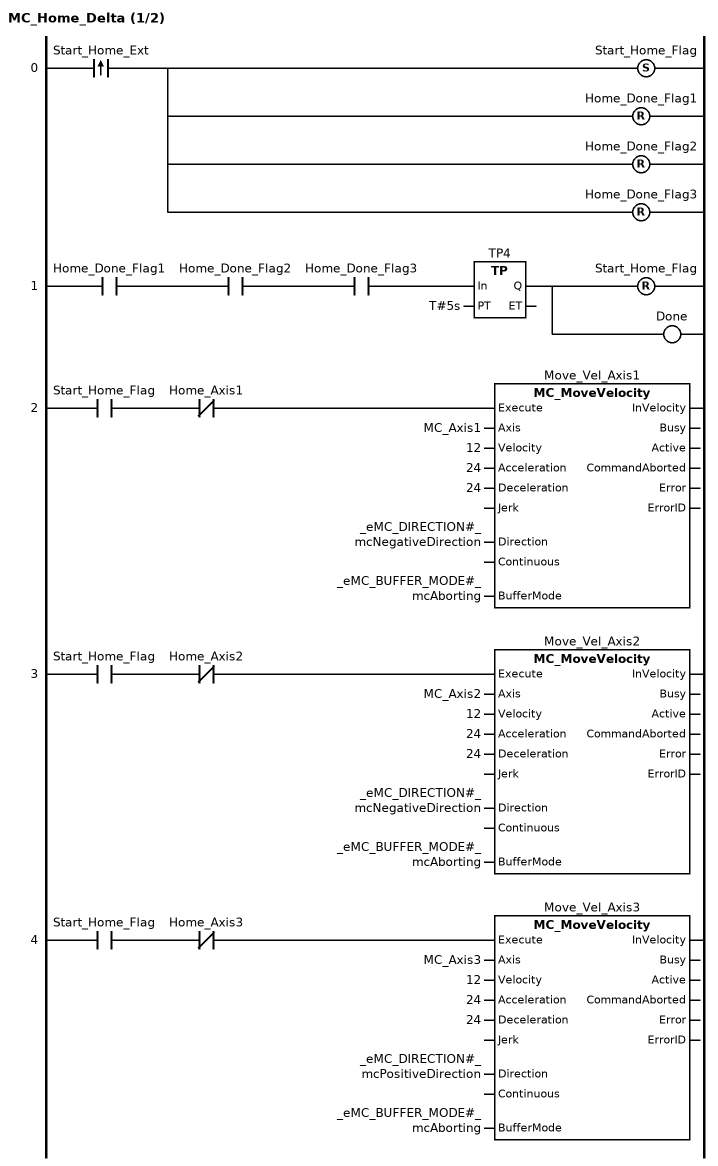
(* Rung 0 *)
_e1(CLK := Start_Home_Ext);
IF _e1.Q THEN
    Start_Home_Flag := TRUE;
    Home_Done_Flag1 := FALSE;
    Home_Done_Flag2 := FALSE;
    Home_Done_Flag3 := FALSE;
END_IF;
(* Rung 1 *)
TP4(In := Home_Done_Flag1 AND Home_Done_Flag2 AND Home_Done_Flag3, PT := T#5s);
IF TP4.Q THEN Start_Home_Flag := FALSE; END_IF;
Done := TP4.Q;
(* Rung 2 *)
Move_Vel_Axis1(Execute := Start_Home_Flag AND NOT Home_Axis1, Axis := MC_Axis1, Velocity := 12, Acceleration := 24, Deceleration := 24, Direction := _eMC_DIRECTION#_mcNegativeDirection, BufferMode := _eMC_BUFFER_MODE#_mcAborting);
(* Rung 3 *)
Move_Vel_Axis2(Execute := Start_Home_Flag AND NOT Home_Axis2, Axis := MC_Axis2, Velocity := 12, Acceleration := 24, Deceleration := 24, Direction := _eMC_DIRECTION#_mcNegativeDirection, BufferMode := _eMC_BUFFER_MODE#_mcAborting);
(* Rung 4 *)
Move_Vel_Axis3(Execute := Start_Home_Flag AND NOT Home_Axis3, Axis := MC_Axis3, Velocity := 12, Acceleration := 24, Deceleration := 24, Direction := _eMC_DIRECTION#_mcPositiveDirection, BufferMode := _eMC_BUFFER_MODE#_mcAborting);

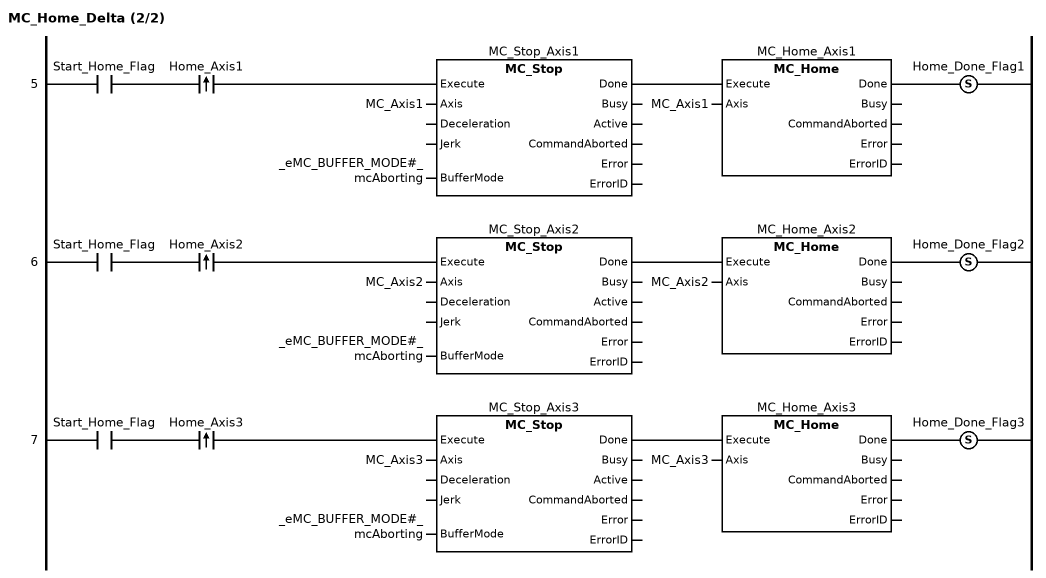
(* Rung 5 *)
_e2(CLK := Home_Axis1);
MC_Stop_Axis1(Execute := Start_Home_Flag AND _e2.Q, Axis := MC_Axis1, BufferMode := _eMC_BUFFER_MODE#_mcAborting);
MC_Home_Axis1(Execute := MC_Stop_Axis1.Done, Axis := MC_Axis1);
IF MC_Home_Axis1.Done THEN Home_Done_Flag1 := TRUE; END_IF;
(* Rung 6 *)
_e3(CLK := Home_Axis2);
MC_Stop_Axis2(Execute := Start_Home_Flag AND _e3.Q, Axis := MC_Axis2, BufferMode := _eMC_BUFFER_MODE#_mcAborting);
MC_Home_Axis2(Execute := MC_Stop_Axis2.Done, Axis := MC_Axis2);
IF MC_Home_Axis2.Done THEN Home_Done_Flag2 := TRUE; END_IF;
(* Rung 7 *)
_e4(CLK := Home_Axis3);
MC_Stop_Axis3(Execute := Start_Home_Flag AND _e4.Q, Axis := MC_Axis3, BufferMode := _eMC_BUFFER_MODE#_mcAborting);
MC_Home_Axis3(Execute := MC_Stop_Axis3.Done, Axis := MC_Axis3);
IF MC_Home_Axis3.Done THEN Home_Done_Flag3 := TRUE; END_IF;
END_FUNCTION_BLOCK

FUNCTION_BLOCK Goto_Absolute
VAR
    Out_Angle1 : LREAL;
    Out_Angle2 : LREAL;
    Out_Angle3 : LREAL;
    Move_abs0 : MC_MoveAbsolute;
    Move_abs1 : MC_MoveAbsolute;
    Move_abs2 : MC_MoveAbsolute;
END_VAR
VAR_INPUT
    Goto_Abs : BOOL;
    X_0 : LREAL;
    Y_0 : LREAL;
    Z_neg300 : LREAL;
END_VAR
VAR_OUTPUT
    Done : BOOL;
END_VAR
VAR_EXTERNAL CONSTANT
    MC_Axis1 : _sAXIS_REF;
    MC_Axis2 : _sAXIS_REF;
    MC_Axis3 : _sAXIS_REF;
END_VAR
VAR
    _t1 : BOOL;
    _e2 : F_TRIG;
END_VAR
(* ladder, written here as Structured Text *)

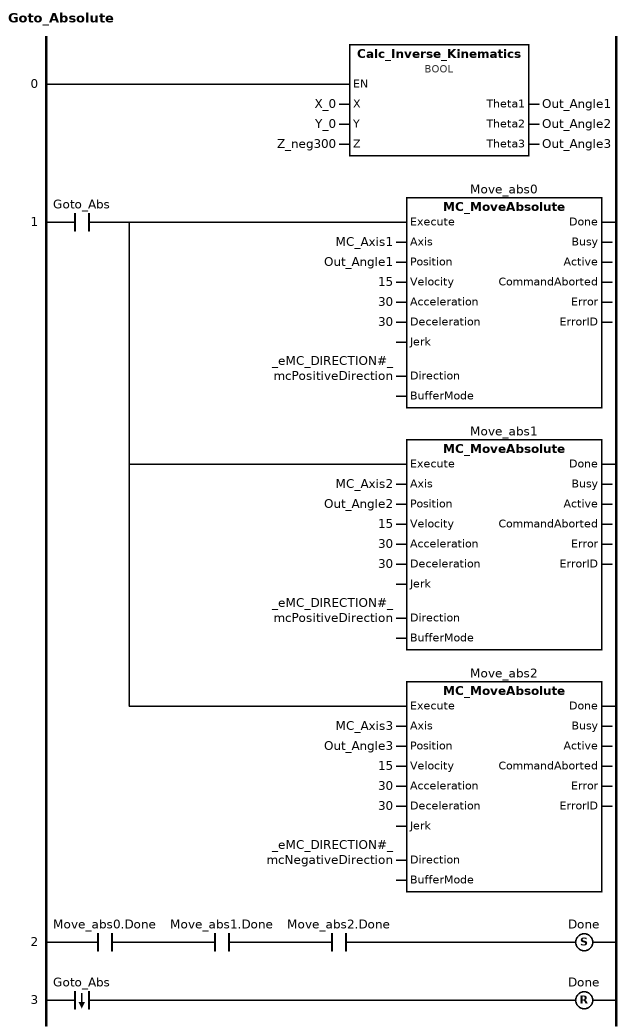
(* Rung 0 *)
_t1 := Calc_Inverse_Kinematics(X := X_0, Y := Y_0, Z := Z_neg300, Theta1 => Out_Angle1, Theta2 => Out_Angle2, Theta3 => Out_Angle3);
(* Rung 1 *)
Move_abs0(Execute := Goto_Abs, Axis := MC_Axis1, Position := Out_Angle1, Velocity := 15, Acceleration := 30, Deceleration := 30, Direction := _eMC_DIRECTION#_mcPositiveDirection);
Move_abs1(Execute := Goto_Abs, Axis := MC_Axis2, Position := Out_Angle2, Velocity := 15, Acceleration := 30, Deceleration := 30, Direction := _eMC_DIRECTION#_mcPositiveDirection);
Move_abs2(Execute := Goto_Abs, Axis := MC_Axis3, Position := Out_Angle3, Velocity := 15, Acceleration := 30, Deceleration := 30, Direction := _eMC_DIRECTION#_mcNegativeDirection);
(* Rung 2 *)
IF Move_abs0.Done AND Move_abs1.Done AND Move_abs2.Done THEN Done := TRUE; END_IF;
(* Rung 3 *)
_e2(CLK := Goto_Abs);
IF _e2.Q THEN Done := FALSE; END_IF;
END_FUNCTION_BLOCK

FUNCTION_BLOCK MC_Inter_Curve_Vel
VAR
    State : INT := 0;
    L : LREAL;
    t_acc : LREAL;
    t_dec : LREAL;
    S_acc : LREAL;
    S_dec : LREAL;
    S_run : LREAL;
    t_run : LREAL;
    T_total : LREAL;
    t : LREAL;
    t_phanh : LREAL;
    S_t : LREAL;
    X_t : LREAL;
    Y_t : LREAL;
    Z_t : LREAL;
    IK_Result : LREAL;
    Check_IK_Error : BOOL;
    tmp_Theta1 : LREAL;
    tmp_Theta2 : LREAL;
    tmp_Theta3 : LREAL;
    MC_Sync_Axis1 : MC_SyncMoveAbsolute;
    MC_Sync_Axis2 : MC_SyncMoveAbsolute;
    MC_Sync_Axis3 : MC_SyncMoveAbsolute;
    Actual_Vmax : LREAL := 100;
    tau : LREAL := 0.2;
    Init_Counter : INT;
    Target_Theta1 : LREAL;
    Target_Theta2 : LREAL;
    Target_Theta3 : LREAL;
    Start_Theta1 : LREAL;
    Start_Theta2 : LREAL;
    Start_Theta3 : LREAL;
    cycle_count : INT;
    Enable_Motion : BOOL;
    MC_SyncMoveAbsolute_Axis1 : MC_SyncMoveAbsolute;
    MC_SyncMoveAbsolute_Axis2 : MC_SyncMoveAbsolute;
    MC_SyncMoveAbsolute_Axis3 : MC_SyncMoveAbsolute;
    Use_Standard_SCurve : BOOL;
    S_limit : LREAL;
    V_reach : LREAL;
    Vec1_X : LREAL;
    Vec1_Y : LREAL;
    Vec1_Z : LREAL;
    Vec2_X : LREAL;
    Vec2_Y : LREAL;
    Vec2_Z : LREAL;
    Len1 : LREAL;
    Len2 : LREAL;
    Cos_Theta : LREAL;
    V_Corner_Max : LREAL;
END_VAR
VAR_INPUT
    X_A : LREAL;
    Y_A : LREAL;
    Z_A : LREAL;
    X_B : LREAL;
    Y_B : LREAL;
    Z_B : LREAL;
    V_max : LREAL;
    A_max : LREAL;
    D_max : LREAL;
END_VAR
VAR_OUTPUT
    Theta1 : LREAL;
    Theta2 : LREAL;
    Theta3 : LREAL;
    Out_Error_IK_OWS : BOOL;
    Busy : BOOL;
END_VAR
VAR_INPUT
    V_Start_Req : LREAL;
END_VAR
VAR_OUTPUT
    Out_Done_Inter : BOOL;
    Out_Done_Blend : BOOL;
    Out_V_End : LREAL;
END_VAR
VAR_INPUT
    Why : BOOL;
    Blend_mode : BOOL;
END_VAR
VAR_IN_OUT
    Execute : BOOL;
END_VAR
VAR_OUTPUT
    t_total_estimate : LREAL;
    Out_T_Segment : LREAL;
END_VAR
VAR_IN_OUT CONSTANT
    Internal_Axis1 : _sAXIS_REF;
    Internal_Axis2 : _sAXIS_REF;
    Internal_Axis3 : _sAXIS_REF;
END_VAR
// ====================================================================
// PHẦN 1: TÍNH TOÁN QUỸ ĐẠO BÊN TRONG STATE MACHINE
// ====================================================================
CASE State OF
    0:  // ================= Step 0: waiting for the new command =================
        IF Execute = TRUE THEN
            Out_Error_IK_OWS := FALSE;  // Reset all fault
            Out_Done_Inter := FALSE;  // Reset interpolation flag
            
            // Cal the inverse kinematic for check
            Check_IK_Error := calc_inverse_kinematics(
                X := X_A, Y := Y_A, Z := Z_A, 
                Theta1 => Target_Theta1, Theta2 => Target_Theta2, Theta3 => Target_Theta3
            );
            
            IF Check_IK_Error = TRUE THEN
                Out_Error_IK_OWS := TRUE; 
                State := 99; 
            ELSE
                Enable_Motion := TRUE;
                // Xoá thời gian của đoạn CŨ. Từ đây tới khi State 1 tính xong,
                // Out_T_Segment = 0 -> caller biết giá trị chưa hợp lệ cho đoạn mới.
                Out_T_Segment := 0.0;

                // LỰA CHỌN LOGIC XUẤT PHÁT DỰA VÀO VẬN TỐC ĐẦU VÀO
                IF V_Start_Req > 0.0 THEN
                    // ĐANG CHẠY NỐI TIẾP (Blend): 
                    // Bỏ qua State 10 làm mượt. Dùng luôn góc lý thuyết Target làm xuất phát để tránh giật
                    Theta1 := Target_Theta1;
                    Theta2 := Target_Theta2;
                    Theta3 := Target_Theta3;
                    State := 1; // Chuyển thẳng sang tính toán S-Curve
                ELSE
                    // XUẤT PHÁT TỪ TRẠNG THÁI DỪNG HẲN: 
                    // Phải lấy vị trí thực tế Act.Pos để chạy mượt 20 chu kỳ triệt tiêu sai số
                    Start_Theta1 := Internal_Axis1.Act.Pos; 
                    Start_Theta2 := Internal_Axis2.Act.Pos;
                    Start_Theta3 := Internal_Axis3.Act.Pos;
                    cycle_count := 1;
                    State := 10; 
                END_IF;
            END_IF;
        ELSE
            // KHI EXECUTE = FALSE
            // Ngắt cờ Blend thành dạng xung (Pulse) để Main Program bắt tín hiệu
            Out_Done_Blend := FALSE; 
            
            Enable_Motion := FALSE; 
            Theta1 := Internal_Axis1.Act.Pos;
            Theta2 := Internal_Axis2.Act.Pos;
            Theta3 := Internal_Axis3.Act.Pos;
        END_IF;

    10: (*
    // =====Step 10: smothing the point start and actual point (from servo) with 20 cyclic time=======
    *)
        IF cycle_count <= 20 THEN
            Theta1 := Start_Theta1 + (Target_Theta1 - Start_Theta1) * (INT_TO_REAL(cycle_count) / 20.0);
            Theta2 := Start_Theta2 + (Target_Theta2 - Start_Theta2) * (INT_TO_REAL(cycle_count) / 20.0);
            Theta3 := Start_Theta3 + (Target_Theta3 - Start_Theta3) * (INT_TO_REAL(cycle_count) / 20.0);
            cycle_count := cycle_count + 1;
        ELSE
            State := 1;
        END_IF;

    1:  // ================= BƯỚC 1: TÍNH TOÁN CẤU HÌNH ĐỘNG LỰC HỌC (S-CURVE/TRAPEZOIDAL) =================
        L := SQRT((X_B - X_A)**2 + (Y_B - Y_A)**2 + (Z_B - Z_A)**2); 

        IF L > 0.0 THEN
            IF Blend_Mode = FALSE THEN
                // --- TRƯỜNG HỢP 1: LÀ ĐIỂM CUỐI CÙNG -> TỰ ĐỘNG PHANH VỀ 0 ---
                Out_V_End := 0.0;
                Use_Standard_SCurve := (V_Start_Req = 0.0); 
                Actual_Vmax := V_max;

                IF Use_Standard_SCurve = TRUE THEN
                    IF L < (0.75 * (Actual_Vmax**2) * (1.0/A_max + 1.0/D_max)) THEN
                        Actual_Vmax := SQRT(L / (0.75 * (1.0/A_max + 1.0/D_max)));
                    END_IF;

                    t_acc := 1.5 * (Actual_Vmax / A_max);
                    t_dec := 1.5 * (Actual_Vmax / D_max);
                    S_acc := 0.5 * Actual_Vmax * t_acc;
                    S_dec := 0.5 * Actual_Vmax * t_dec;
                    S_run := L - S_acc - S_dec;
                    t_run := S_run / Actual_Vmax;
                    T_total := t_acc + t_run + t_dec;
                ELSE
                    S_limit := (ABS(Actual_Vmax**2 - V_Start_Req**2)/(2.0*A_max)) + (ABS(Actual_Vmax**2)/(2.0*D_max));
                    IF S_limit > L THEN
                        Actual_Vmax := SQRT((2.0*A_max*D_max*L + D_max*(V_Start_Req**2)) / (A_max + D_max));
                    END_IF;

                    t_acc := ABS(Actual_Vmax - V_Start_Req) / A_max;
                    t_dec := ABS(Actual_Vmax) / D_max; 
                    S_acc := (V_Start_Req + Actual_Vmax) * 0.5 * t_acc;
                    S_dec := Actual_Vmax * 0.5 * t_dec;
                    S_run := L - S_acc - S_dec;
                    
                    IF S_run < 0.0 THEN S_run := 0.0; END_IF;
                    t_run := S_run / Actual_Vmax;
                    T_total := t_acc + t_run + t_dec;
                END_IF;

            ELSE
                // --- TRƯỜNG HỢP 2: CHẠY NỐI TIẾP (BLEND) ---
                Use_Standard_SCurve := FALSE;

                // Blend mode: giữ vận tốc cao, không giảm tốc ở điểm B
                Out_V_End := V_max;

                // Tính toán cấu hình hình thang (Tăng tốc - Chạy đều)
                Actual_Vmax := V_max;
                S_limit := (ABS(Actual_Vmax**2 - V_Start_Req**2)/(2.0*A_max)) + (ABS(Actual_Vmax**2 - Out_V_End**2)/(2.0*D_max));

                IF S_limit > L THEN
                    // Không đủ quãng đường để đạt V_max
                    Actual_Vmax := SQRT((2.0*A_max*D_max*L + D_max*(V_Start_Req**2) + A_max*(Out_V_End**2)) / (A_max + D_max));
                END_IF;

                t_acc := ABS(Actual_Vmax - V_Start_Req) / A_max;
                t_dec := ABS(Actual_Vmax - Out_V_End) / D_max;

                S_acc := (V_Start_Req + Actual_Vmax) * 0.5 * t_acc;
                S_dec := (Out_V_End + Actual_Vmax) * 0.5 * t_dec;
                S_run := L - S_acc - S_dec;

                IF S_run < 0.0 THEN S_run := 0.0; END_IF;
                t_run := S_run / Actual_Vmax;
                T_total := t_acc + t_run + t_dec;
            END_IF;

            // Thời gian ước tính của ĐOẠN NÀY -> caller cộng dồn thành tổng quỹ đạo
            // và dùng làm gốc tính thời điểm nhả vật của bơm.
            Out_T_Segment := T_total;

            t := 0.0;
            State := 2;
        ELSE
            Execute := FALSE;
            State := 0;
        END_IF;

    2:  // ================= BƯỚC 2: NỘI SUY TỌA ĐỘ THEO THỜI GIAN =================
        IF t <= T_total THEN
            // 2.1 Tính quãng đường S_t
            IF Use_Standard_SCurve = TRUE THEN
                IF t <= t_acc THEN
                    tau := t / t_acc; 
                    S_t := Actual_Vmax * t_acc * ((tau ** 3) - 0.5 * (tau ** 4));
                ELSIF t <= (t_acc + t_run) THEN
                    S_t := S_acc + Actual_Vmax * (t - t_acc);
                ELSE
                    t_phanh := t - (t_acc + t_run);
                    tau := t_phanh / t_dec; 
                    S_t := S_acc + S_run + Actual_Vmax * t_dec * (tau - (tau ** 3) + 0.5 * (tau ** 4));
                END_IF;
            ELSE
                IF t <= t_acc THEN
                    S_t := V_Start_Req * t + 0.5 * A_max * (t**2);
                ELSIF t <= (t_acc + t_run) THEN
                    S_t := S_acc + Actual_Vmax * (t - t_acc);
                ELSE
                    t_phanh := t - (t_acc + t_run);
                    S_t := S_acc + S_run + Actual_Vmax * t_phanh - 0.5 * D_max * (t_phanh**2);
                END_IF;
                
                IF S_t > L THEN S_t := L; END_IF; 
            END_IF;

            // 2.2 Tính tọa độ Descartes X, Y, Z tại S_t
            X_t := X_A + (S_t / L) * (X_B - X_A);
            Y_t := Y_A + (S_t / L) * (Y_B - Y_A);
            Z_t := Z_A + (S_t / L) * (Z_B - Z_A);

            // 2.3 Giải Động Học Nghịch (IK) để tìm góc cho 3 trục
            Check_IK_Error := calc_inverse_kinematics(
                X := X_t, Y := Y_t, Z := Z_t, 
                Theta1 => tmp_Theta1, Theta2 => tmp_Theta2, Theta3 => tmp_Theta3
            );
            
            IF Check_IK_Error = TRUE THEN
                Out_Error_IK_OWS := TRUE; 
                State := 99; 
                RETURN; 
            END_IF;

            // Cập nhật vị trí đẩy xuống lệnh gọi Servo
            Theta1 := tmp_Theta1;
            Theta2 := tmp_Theta2;
            Theta3 := tmp_Theta3;

            t := t + 0.004; // Chu kỳ lấy mẫu nội suy (4ms)

        ELSE
            // ================= KẾT THÚC ĐOẠN ĐƯỜNG (HẾT THỜI GIAN T_total) =================
            IF (Blend_Mode = TRUE) AND (Out_V_End > 0.0) THEN
                // CHẠY NỐI TIẾP: Bật cờ Blend, chờ nhả Execute
                Out_Done_Blend := TRUE; 
                Execute := FALSE; 
                State := 0; // Quay về State 0 chực chờ nạp điểm mới và nội suy tiếp
            ELSE
                // DỪNG HẲN: Chuyển sang State 3 đợi Servo Settle
                State := 3; 
            END_IF;
        END_IF;

    3:  // ================= BƯỚC 3: KIỂM TRA SAI SỐ DỪNG (SETTLE) =================
        Enable_Motion := FALSE; 
        
        // Đọc ACT.POS để xác nhận Servo đã bám sát điểm đích với sai số < 0.0005 độ
        IF (ABS(Theta1 - Internal_Axis1.Act.Pos) <= 0.0005) AND 
           (ABS(Theta2 - Internal_Axis2.Act.Pos) <= 0.0005) AND 
           (ABS(Theta3 - Internal_Axis3.Act.Pos) <= 0.0005)
           THEN
            Out_Done_Inter := TRUE;
        ELSE
            Out_Done_Inter := FALSE;
        END_IF;

        // Xả cờ và reset State khi Servo báo hết Busy
        IF (MC_Sync_Axis1.Busy = FALSE) AND 
           (MC_Sync_Axis2.Busy = FALSE) AND 
           (MC_Sync_Axis3.Busy = FALSE) THEN
            
            Execute := FALSE;  
            State := 0;        
        END_IF;

    99: // ================= BƯỚC 99: LỖI KINEMATICS =================
        Execute := FALSE;
        Enable_Motion := FALSE; 
        IF Out_Error_IK_OWS = FALSE THEN
             State := 0;
        END_IF;
END_CASE;

// ====================================================================
// PHẦN 2: GỌI HÀM SERVO (LUÔN ĐƯỢC QUÉT Ở CUỐI CHU KỲ)
// ====================================================================
// Sử dụng hàm đồng bộ vị trí, servo sẽ bám theo biến Theta liên tục
MC_Sync_Axis1(Axis := Internal_Axis1, Execute := Enable_Motion, Position := Theta1);
MC_Sync_Axis2(Axis := Internal_Axis2, Execute := Enable_Motion, Position := Theta2);
MC_Sync_Axis3(Axis := Internal_Axis3, Execute := Enable_Motion, Position := Theta3);
END_FUNCTION_BLOCK

FUNCTION_BLOCK FB_TeachingMode
VAR
    Pw_Power_0 : MC_Power;
    Pw_Power_1 : MC_Power;
    Pw_Power_2 : MC_Power;
    Pw_servo_on : BOOL := True;
    button_teaching_old : BOOL := False;
    button_teaching_fall : BOOL := False;
    start_teaching_mode_old : BOOL := False;
    fk_err : BOOL := False;
END_VAR
VAR_INPUT
    start_teaching_mode : BOOL;
    button_teaching : BOOL;
END_VAR
VAR_OUTPUT
    theta_teaching1 : LREAL;
    theta_teaching2 : LREAL;
    theta_teaching3 : LREAL;
    pos_teaching1 : LREAL;
    pos_teaching2 : LREAL;
    pos_teaching3 : LREAL;
    teaching_done : BOOL;
    teaching_err : BOOL;
END_VAR
VAR_IN_OUT CONSTANT
    inter_MC_Axis1 : _sAXIS_REF;
    inter_MC_Axis2 : _sAXIS_REF;
    inter_MC_Axis3 : _sAXIS_REF;
END_VAR
// =========================================================================================
// FUNCTION_BLOCK: FB_TeachingMode
// =========================================================================================

// -----------------------------------------------------------------------------------------
// Reset xung báo mỗi chu kỳ quét
// -----------------------------------------------------------------------------------------
teaching_done := FALSE;
teaching_err  := FALSE;

// -----------------------------------------------------------------------------------------
// Sườn lên của start_teaching_mode: vừa VÀO Teaching Mode
// -> tránh bắt sườn giả nếu button_teaching đã lỡ giữ sẵn từ trước khi vào mode
// -----------------------------------------------------------------------------------------
IF start_teaching_mode AND NOT start_teaching_mode_old THEN
    button_teaching_old := button_teaching;
END_IF;
start_teaching_mode_old := start_teaching_mode;

IF start_teaching_mode THEN

    // 1. Bắt sườn xuống của nút button_teaching (khoảnh khắc vừa nhả tay)
    button_teaching_fall := NOT button_teaching AND button_teaching_old;
    button_teaching_old  := button_teaching;

    // 2. Điều khiển nguồn Servo theo trạng thái nút
    IF button_teaching THEN
        // Giữ nút: tắt mô-men Servo, thắng NC 24V đang mở sẵn -> kéo tay tự do
        Pw_servo_on := FALSE;
    ELSE
        // Thả nút: bật Servo ON để khóa giữ vị trí ngay lập tức
        Pw_servo_on := TRUE;
    END_IF;

    // 3. Ghi nhận điểm dạy khi vừa thả nút (sườn xuống)
    IF button_teaching_fall THEN

        // a. Đọc chính xác góc Encoder thực tế 3 trục tại thời điểm vừa nhả tay (độ)
        theta_teaching1 := inter_MC_Axis1.Act.Pos;
        theta_teaching2 := inter_MC_Axis2.Act.Pos;
        theta_teaching3 := inter_MC_Axis3.Act.Pos;

        // b. Gọi Động Học Thuận (Forward Kinematics) để tính tọa độ Cartesian (X, Y, Z)
        fk_err := Calc_Forward_Kinematic(
            EN        := TRUE,
            Theta1    := theta_teaching1,
            Theta2    := theta_teaching2,
            Theta3    := theta_teaching3,
            Calc_OutX => pos_teaching1,
            Calc_OutY => pos_teaching2,
            Calc_OutZ => pos_teaching3
        );

        // c. Báo kết quả cho caller (Program_Main) qua xung teaching_done / teaching_err
        IF fk_err THEN
            teaching_err := TRUE;
        ELSE
            teaching_done := TRUE;
        END_IF;

    END_IF;

ELSE
    // Ngoài Teaching Mode: luôn giữ Servo ON, không cho button_teaching có tác dụng
    Pw_servo_on := TRUE;
    button_teaching_fall := FALSE;
    button_teaching_old  := button_teaching; // tránh sườn giả khi vào lại mode lần sau
END_IF;

// 4. Thực thi khối điều khiển MC_Power cho 3 trục Delta (chạy mọi scan)
Pw_Power_0(Axis := inter_MC_Axis1, Enable := Pw_servo_on);
Pw_Power_1(Axis := inter_MC_Axis2, Enable := Pw_servo_on);
Pw_Power_2(Axis := inter_MC_Axis3, Enable := Pw_servo_on);
END_FUNCTION_BLOCK

FUNCTION_BLOCK FB_ICV_Sequencer
VAR
    ICV_Run : MC_Inter_Curve_Vel;
    State : INT;
    Last_Idx : INT;
    Idx_Max : DINT;
    Exec_Prev : BOOL;
    Exec_Edge : BOOL;
    Blend_Prev : BOOL;
    Blend_Edge : BOOL;
    Inter_Prev : BOOL;
    Inter_Edge : BOOL;
    Seq_Exec : BOOL;
    Seq_Load : BOOL;
    Seq_Blend : BOOL;
    Seq_X_A : LREAL;
    Seq_Y_A : LREAL;
    Seq_Z_A : LREAL;
    Seq_X_B : LREAL;
    Seq_Y_B : LREAL;
    Seq_Z_B : LREAL;
    Seq_V_Start : LREAL;
    i : INT;
END_VAR
VAR_INPUT
    Execute : BOOL;
    Max_Index : INT;
    Abort : BOOL;
    ErrReset : BOOL;
    N_Points : INT;
    V_max : LREAL;
    A_max : LREAL;
    D_max : LREAL;
END_VAR
VAR_IN_OUT
    Pos_X : ARRAY[*] OF LREAL;
    Pos_Y : ARRAY[*] OF LREAL;
    Pos_Z : ARRAY[*] OF LREAL;
    T_Seg : ARRAY[*] OF LREAL;
END_VAR
VAR_IN_OUT CONSTANT
    Int_Axis1 : _sAXIS_REF;
    Int_Axis2 : _sAXIS_REF;
    Int_Axis3 : _sAXIS_REF;
END_VAR
VAR_OUTPUT
    Busy : BOOL;
    Done : BOOL;
    Error : BOOL;
    ErrorID : INT;
    SegIdx : INT;
    IsLastSeg : BOOL;
    T_Total : LREAL;
    T_SegNow : LREAL;
END_VAR
// =====================================================================================
// FUNCTION_BLOCK: FB_ICV_Sequencer
// Chạy quỹ đạo N điểm bằng DUY NHẤT 1 instance MC_Inter_Curve_Vel bên trong.
// Thay thế toàn bộ Rung 13..18 (6 FB nối cứng) của bản cũ.
//
//   N điểm  ->  N-1 đoạn  ->  chỉ số đoạn SegIdx = 0 .. (N_Points - 2)
//   Đoạn i  :  Pos[i] -> Pos[i+1]
//   Blend   :  TRUE với i < N_Points-2 ; FALSE với đoạn cuối (phanh về 0)
//   V_Start :  0.0 với i = 0 ; = Out_V_End của đoạn trước với i > 0
//
// FB này CHỈ lo quỹ đạo. Không đụng tới bơm/van — caller tự làm, dùng 3 output
// SegIdx / IsLastSeg / T_SegNow. Nhờ vậy FB dùng lại được cho máy khác.
//
// ---------------------------------------------------------------------------------
// BẢNG KHAI BÁO (gõ vào tab khai báo của FB trong Sysmac Studio)
// ---------------------------------------------------------------------------------
// VAR_INPUT
//     Execute    : BOOL;      // SƯỜN LÊN = chạy quỹ đạo mới
//     Abort      : BOOL;      // huỷ ngay lập tức
//     ErrReset   : BOOL;      // xoá lỗi, đưa FB về IDLE
//     N_Points   : INT;       // SỐ ĐIỂM (không phải số đoạn)
//     Max_Index  : INT;       // chỉ số LỚN NHẤT của mảng Pos_X (31 nếu ARRAY[0..31])
//     V_max      : LREAL;
//     A_max      : LREAL;
//     D_max      : LREAL;
// END_VAR
//
// VAR_IN_OUT                              // ARRAY[*] = truyền THAM CHIẾU, không copy
//     Pos_X      : ARRAY[*] OF LREAL;     // toạ độ X, PHẢI đánh chỉ số từ 0
//     Pos_Y      : ARRAY[*] OF LREAL;     // toạ độ Y
//     Pos_Z      : ARRAY[*] OF LREAL;     // toạ độ Z
//     T_Seg      : ARRAY[*] OF LREAL;     // FB GHI thời gian từng đoạn ra đây
//     Int_Axis1  : _sAXIS_REF;            // BẮT BUỘC In/Out ở MỌI TẦNG
//     Int_Axis2  : _sAXIS_REF;            // Đặt tên Int_* để phân biệt với biến global
//     Int_Axis3  : _sAXIS_REF;            // MC_Axis* của trục thật bên ngoài
// END_VAR
//
// CHUỖI TRUYỀN TRỤC - chỉ cần 1 tầng khai sai là gãy cả chuỗi:
//
//   Program_Main          ICV_Sequencer          MC_Inter_Curve_Vel      MC_Sync_Axis*
//   MC_Axis1  ────────►   Int_Axis1  ────────►   Internal_Axis1  ────►   Axis
//   (global thật)         (In/Out)               (In/Out)                (yêu cầu Omron)
//
//   Ở Program_Main:   Traj( Int_Axis1 := MC_Axis1, ... )
//   Ở FB này:         ICV_Run( Internal_Axis1 := Int_Axis1, ... )
//                                    ▲                ▲
//                                    │                └── biến In/Out của FB này
//                                    └── tên tham số của MC_Inter_Curve_Vel
//
// MC_Inter_Curve_Vel PHẢI khai 3 trục ở tab In/Out. Nếu để ở tab Externals thì nó
// không có chân tham số -> lời gọi dưới đây báo
//   "The variable 'MC_Axis1' is not an in-out variable"
// và lỗi sẽ trỏ vào TÊN THAM SỐ bên TRÁI dấu := (cột 5), không phải argument.
//
// VAR_OUTPUT
//     Busy       : BOOL;      // đang chạy quỹ đạo
//     Done       : BOOL;      // XUNG 1 SCAN: xong cả quỹ đạo, servo đã settle
//     Error      : BOOL;      // có lỗi, FB đứng yên chờ ErrReset
//     ErrorID    : INT;       // 1 = N_Points sai/mảng quá nhỏ ; 2 = IK ngoài vùng
//     SegIdx     : INT;       // đang chạy đoạn thứ mấy (0 .. N_Points-2)
//     IsLastSeg  : BOOL;      // TRUE khi đang ở đoạn cuối -> caller dùng cho bơm
//     T_Total    : LREAL;     // TỔNG thời gian cộng dồn (giây)
//     T_SegNow   : LREAL;     // thời gian đoạn đang chạy (0 = chưa tính xong)
// END_VAR
//
// VAR
//     ICV_Run    : MC_Inter_Curve_Vel;    // 1 instance DUY NHẤT
//     State      : INT;                   // 0=idle 1=running 2=done 9=error
//     Last_Idx   : INT;                   // chỉ số đoạn cuối = N_Points - 2
//     Exec_Prev  : BOOL;
//     Exec_Edge  : BOOL;
//     Blend_Prev : BOOL;
//     Blend_Edge : BOOL;
//     Inter_Prev : BOOL;
//     Inter_Edge : BOOL;
//     Seq_Exec   : BOOL;
//     Seq_Load   : BOOL;
//     Seq_Blend  : BOOL;
//     Seq_X_A    : LREAL;
//     Seq_Y_A    : LREAL;
//     Seq_Z_A    : LREAL;
//     Seq_X_B    : LREAL;
//     Seq_Y_B    : LREAL;
//     Seq_Z_B    : LREAL;
//     Seq_V_Start: LREAL;
//     i          : INT;
// END_VAR
//
// ---------------------------------------------------------------------------------
// THỨ TỰ 7 KHỐI DƯỚI ĐÂY LÀ BẮT BUỘC
//   (1) xoá xung -> (2) GỌI FB NỘI SUY -> (3) bắt sườn -> (4) abort
//   -> (5) state machine -> (6) nạp đoạn kế -> (7) xuất output
// Vì (2) đứng TRƯỚC (5)(6): đoạn i vừa xong thì đoạn i+1 được nạp NGAY trong cùng
// chu kỳ quét -> thời gian chuyển đoạn bằng đúng kiến trúc 6-FB cũ, không chậm thêm.
// =====================================================================================


// -------------------------------------------------------------------------------------
// (1) XUNG 1 SCAN: XOÁ Ở ĐẦU CHU KỲ
// -------------------------------------------------------------------------------------
Done := FALSE;


// -------------------------------------------------------------------------------------
// (2) GỌI FB NỘI SUY  (1 instance duy nhất, dùng lại cho mọi đoạn)
//     Execute của ICV_Run là VAR_IN_OUT: nó tự hạ Seq_Exec khi chạy xong 1 đoạn.
// -------------------------------------------------------------------------------------
ICV_Run(
    Execute     := Seq_Exec,
    X_A         := Seq_X_A,
    Y_A         := Seq_Y_A,
    Z_A         := Seq_Z_A,
    X_B         := Seq_X_B,
    Y_B         := Seq_Y_B,
    Z_B         := Seq_Z_B,
    V_Start_Req := Seq_V_Start,
    V_max       := V_max,
    A_max       := A_max,
    D_max       := D_max,
    Blend_Mode  := Seq_Blend,
    // TRÁI  = tên tham số của MC_Inter_Curve_Vel  (Internal_AxisN)
    // PHẢI  = biến In/Out của FB này              (Int_AxisN)
    Internal_Axis1 := Int_Axis1,
    Internal_Axis2 := Int_Axis2,
    Internal_Axis3 := Int_Axis3
);


// -------------------------------------------------------------------------------------
// (3) BẮT SƯỜN LÊN
//     Out_Done_Blend BẮT BUỘC dùng sườn, KHÔNG dùng mức. Lý do: khi ta nạp đoạn kế
//     ngay lập tức, Seq_Exec lên TRUE trở lại nên nhánh ELSE của State 0 trong ICV_Run
//     (nơi nó tự hạ Out_Done_Blend) không bao giờ chạy -> cờ giữ mức TRUE suốt quỹ đạo.
//     Dùng mức sẽ nhảy đoạn mỗi 4 ms và đốt hết waypoint trong ~50 ms.
// -------------------------------------------------------------------------------------
Blend_Edge := ICV_Run.Out_Done_Blend AND NOT Blend_Prev;
Blend_Prev := ICV_Run.Out_Done_Blend;

Inter_Edge := ICV_Run.Out_Done_Inter AND NOT Inter_Prev;
Inter_Prev := ICV_Run.Out_Done_Inter;

Exec_Edge  := Execute AND NOT Exec_Prev;
Exec_Prev  := Execute;


// -------------------------------------------------------------------------------------
// (4) ABORT
// -------------------------------------------------------------------------------------
IF Abort THEN
    Seq_Exec := FALSE;
    Seq_Load := FALSE;
    Busy     := FALSE;
    State    := 0;
END_IF;


// -------------------------------------------------------------------------------------
// (5) MÁY TRẠNG THÁI
// -------------------------------------------------------------------------------------
CASE State OF

    0:  // ============ IDLE: chờ sườn lên của Execute ============
        Busy     := FALSE;
        Seq_Exec := FALSE;

        IF Exec_Edge THEN

            // Max_Index = chỉ số LỚN NHẤT của mảng Pos_X, do caller truyền vào
            // (31 nếu khai ARRAY[0..31]). Không dùng UpperBound vì bản Sysmac này
            // không có lệnh đó.
            // N điểm cần chỉ số 0..N-1, nên N-1 phải <= Max_Index.
            IF (N_Points < 2) OR ((N_Points - 1) > Max_Index) THEN
                // Số điểm vô lý, hoặc mảng không đủ chỗ -> chặn trước khi động cơ chạy
                Error   := TRUE;
                ErrorID := 1;
                State   := 9;
            ELSE
                Error   := FALSE;
                ErrorID := 0;

                // Chốt chỉ số đoạn cuối NGAY LÚC NÀY. Nếu caller lỡ đổi N_Points
                // giữa chừng thì quỹ đạo đang chạy vẫn dùng giá trị cũ -> an toàn.
                Last_Idx := N_Points - 2;

                // Reset bộ đếm thời gian của lượt chạy mới
                T_Total := 0.0;
                // T_Seg nhỏ hơn Pos_X đúng 1 phần tử: 32 điểm -> 31 đoạn
                FOR i := 0 TO (Max_Index - 1) DO
                    T_Seg[i] := 0.0;
                END_FOR;

                SegIdx      := 0;
                Seq_V_Start := 0.0;         // đoạn đầu luôn xuất phát từ dừng
                Seq_Load    := TRUE;        // -> khối (6) nạp Pos[0] -> Pos[1]
                Busy        := TRUE;
                State       := 1;
            END_IF;
        END_IF;


    1:  // ============ RUNNING: đang chạy đoạn SegIdx ============
        IF ICV_Run.Out_Error_IK_OWS THEN
            // Điểm nằm ngoài vùng làm việc -> dừng cả quỹ đạo
            Error    := TRUE;
            ErrorID  := 2;
            Seq_Exec := FALSE;
            State    := 9;

        ELSIF Blend_Edge THEN
            // --- Đoạn SegIdx vừa xong ở chế độ NỐI TIẾP ---
            // Out_T_Segment vẫn giữ T_total của đoạn vừa xong (ICV_Run chỉ xoá nó ở
            // State 0 của đoạn kế, tức chu kỳ sau) -> đọc ở đây là chính xác.
            T_Seg[SegIdx] := ICV_Run.Out_T_Segment;
            T_Total       := T_Total + T_Seg[SegIdx];

            Seq_V_Start   := ICV_Run.Out_V_End;   // NỐI VẬN TỐC: V_end(i) -> V_start(i+1)
            SegIdx        := SegIdx + 1;
            Seq_Load      := TRUE;                // -> khối (6) nạp đoạn kế

        ELSIF Inter_Edge THEN
            // --- Đoạn CUỐI vừa dừng hẳn và servo đã bám đúng đích ---
            T_Seg[SegIdx] := ICV_Run.Out_T_Segment;
            T_Total       := T_Total + T_Seg[SegIdx];

            Seq_Exec      := FALSE;
            State         := 2;
        END_IF;


    2:  // ============ DONE ============
        Busy  := FALSE;
        Done  := TRUE;                      // xung 1 scan
        State := 0;


    9:  // ============ ERROR: đứng yên chờ ErrReset ============
        Busy     := FALSE;
        Seq_Exec := FALSE;
        IF ErrReset THEN
            Error   := FALSE;
            ErrorID := 0;
            State   := 0;
        END_IF;

END_CASE;


// -------------------------------------------------------------------------------------
// (6) NẠP ĐOẠN HIỆN TẠI  (Pos[SegIdx] -> Pos[SegIdx + 1])
//     Chạy SAU máy trạng thái để dùng đúng SegIdx vừa tăng.
// -------------------------------------------------------------------------------------
IF Seq_Load THEN
    Seq_Load := FALSE;

    Seq_X_A := Pos_X[SegIdx];
    Seq_Y_A := Pos_Y[SegIdx];
    Seq_Z_A := Pos_Z[SegIdx];

    Seq_X_B := Pos_X[SegIdx + 1];
    Seq_Y_B := Pos_Y[SegIdx + 1];
    Seq_Z_B := Pos_Z[SegIdx + 1];

    // Đoạn cuối có chỉ số Last_Idx (= N_Points - 2) -> Blend = FALSE -> phanh về 0.
    // N_Points = 7: đoạn 0..4 Blend=TRUE, đoạn 5 Blend=FALSE.
    // N_Points = 2: chỉ có đoạn 0, (0 < 0) = FALSE -> phanh luôn. Đúng.
    Seq_Blend := (SegIdx < Last_Idx);

    Seq_Exec := TRUE;
END_IF;


// -------------------------------------------------------------------------------------
// (7) XUẤT OUTPUT PHỤ TRỢ CHO CALLER
//     Caller dùng 2 cái này để điều khiển bơm/van mà không cần biết ruột FB.
// -------------------------------------------------------------------------------------
IsLastSeg := Busy AND (SegIdx = Last_Idx);
T_SegNow  := ICV_Run.Out_T_Segment;
END_FUNCTION_BLOCK